KUKA KRL program: MyProgram_266().src

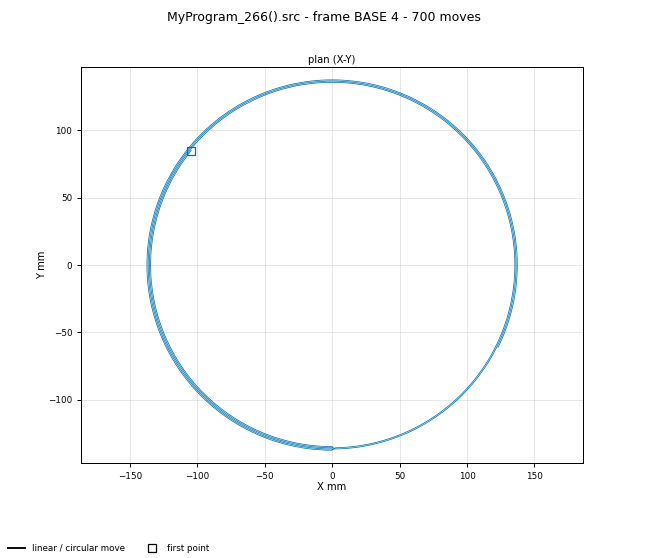
[picture p0: tool path of MyProgram_266().src in frame BASE 4, 700 of 700 moves have a stored position in this frame; points joined in program order, loops and branches not executed]
&ACCESS RVP
&REL 1
&PARAM TEMPLATE = C:\KRC\Roboter\Template\vorgabe
&PARAM EDITMASK = *
DEF MyProgram_266()
; ---- Setting reference (Base) ----
$BASE = BASE_DATA[4]

; --------------------------
; ---- Setting tool (TCP) ----
$TOOL = TOOL_DATA[3]
; --------------------------

$VEL.CP = VEL_APROX_PRINT
Startdeposition()
$VEL.CP = VEL_PRINT
LIN {X -104.4746,Y 84.848,Z 169,A 141.9621,B 9.8477,C 0.0918,E1 9.7233,E2 309.1377} C_DIS
LIN {X -107.2556,Y 81.3036,Z 169,A 143.6702,B 9.8476,C 0.1001,E1 9.7204,E2 307.4569} C_DIS
LIN {X -111.5663,Y 75.2791,Z 169,A 147.0659,B 9.8476,C 0.1033,E1 9.7149,E2 304.0355} C_DIS
LIN {X -114.0415,Y 71.475,Z 169,A 148.9826,B 9.8475,C 0.1084,E1 9.712,E2 302.1227} C_DIS
LIN {X -115.8284,Y 68.5413,Z 169,A 150.5259,B 9.8475,C 0.1107,E1 9.7098,E2 300.5712} C_DIS
LIN {X -118.6938,Y 63.4493,Z 169,A 153.1021,B 9.8474,C 0.1155,E1 9.7063,E2 297.9869} C_DIS
LIN {X -120.5086,Y 59.9271,Z 169,A 154.6631,B 9.8474,C 0.1222,E1 9.7043,E2 296.4429} C_DIS
LIN {X -122.0379,Y 56.7472,Z 169,A 156.1056,B 9.8473,C 0.1272,E1 9.7026,E2 295.0093} C_DIS
LIN {X -123.501,Y 53.4877,Z 169,A 157.6774,B 9.8473,C 0.1304,E1 9.7009,E2 293.4329} C_DIS
LIN {X -124.8461,Y 50.2682,Z 169,A 159.1832,B 9.8472,C 0.1341,E1 9.6993,E2 291.9263} C_DIS
LIN {X -126.2668,Y 46.5893,Z 169,A 161.0061,B 9.8472,C 0.1361,E1 9.6974,E2 290.0877} C_DIS
LIN {X -127.5662,Y 42.9007,Z 169,A 162.6082,B 9.8471,C 0.1419,E1 9.696,E2 288.495} C_DIS
LIN {X -128.6173,Y 39.6372,Z 169,A 164.0174,B 9.847,C 0.1468,E1 9.6948,E2 287.0935} C_DIS
LIN {X -129.8851,Y 35.2642,Z 169,A 166.1874,B 9.847,C 0.1482,E1 9.6932,E2 284.8975} C_DIS
LIN {X -130.8817,Y 31.3605,Z 169,A 168.0934,B 9.847,C 0.1497,E1 9.6919,E2 282.97} C_DIS
LIN {X -131.6037,Y 28.1781,Z 169,A 169.2729,B 9.8468,C 0.1574,E1 9.6912,E2 281.8174} C_DIS
LIN {X -132.3186,Y 24.6117,Z 169,A 171.627,B 9.847,C 0.1475,E1 9.69,E2 279.3666} C_DIS
LIN {X -133.2931,Y 18.6182,Z 169,A 173.4883,B 9.8466,C 0.1679,E1 9.6893,E2 277.5966} C_DIS
LIN {X -133.7452,Y 15.0386,Z 169,A 175.0197,B 9.8466,C 0.1725,E1 9.6887,E2 276.0674} C_DIS
LIN {X -134.1082,Y 11.3371,Z 169,A 176.5691,B 9.8465,C 0.1777,E1 9.6884,E2 274.5236} C_DIS
LIN {X -134.3787,Y 7.5153,Z 169,A 178.3708,B 9.8465,C 0.1794,E1 9.688,E2 272.7028} C_DIS
LIN {X -134.5281,Y 3.9764,Z 169,A 179.8134,B 9.8463,C 0.1849,E1 9.688,E2 271.2696} C_DIS
LIN {X -134.589,Y -0.2836,Z 169,A -178.249,B 9.8463,C 0.188,E1 9.6879,E2 269.3188} C_DIS
LIN {X -134.5104,Y -4.577,Z 169,A -176.4181,B 9.8462,C 0.1933,E1 9.688,E2 267.4893} C_DIS
LIN {X -134.2976,Y -8.8324,Z 169,A -174.5756,B 9.8461,C 0.1981,E1 9.6883,E2 265.6449} C_DIS
LIN {X -133.9649,Y -12.9206,Z 169,A -172.93,B 9.846,C 0.2049,E1 9.6887,E2 264.0132} C_DIS
LIN {X -133.5317,Y -16.8296,Z 169,A -171.2069,B 9.8459,C 0.2089,E1 9.6893,E2 262.2858} C_DIS
LIN {X -133.1154,Y -19.8582,Z 169,A -169.0696,B 9.8461,C 0.1976,E1 9.6903,E2 260.0468} C_DIS
LIN {X -132.0948,Y -25.7822,Z 169,A -167.1873,B 9.8457,C 0.2171,E1 9.6912,E2 258.2501} C_DIS
LIN {X -131.1442,Y -30.2452,Z 169,A -165.035,B 9.8457,C 0.2188,E1 9.6925,E2 256.0738} C_DIS
LIN {X -130.3652,Y -33.4442,Z 169,A -163.6911,B 9.8455,C 0.2238,E1 9.6934,E2 254.7381} C_DIS
LIN {X -129.1038,Y -38.0226,Z 169,A -161.8309,B 9.8454,C 0.2323,E1 9.6948,E2 252.8994} C_DIS
LIN {X -127.7896,Y -42.2298,Z 169,A -159.9505,B 9.8452,C 0.2374,E1 9.6964,E2 251.02} C_DIS
LIN {X -126.6409,Y -45.5579,Z 169,A -158.4535,B 9.8452,C 0.2415,E1 9.6978,E2 249.5244} C_DIS
LIN {X -125.6224,Y -48.298,Z 169,A -157.1558,B 9.8451,C 0.2439,E1 9.6991,E2 248.2211} C_DIS
LIN {X -124.3665,Y -51.4452,Z 169,A -155.6269,B 9.8451,C 0.2462,E1 9.7007,E2 246.6826} C_DIS
LIN {X -123.0232,Y -54.5791,Z 169,A -153.402,B 9.8453,C 0.2358,E1 9.7034,E2 244.363} C_DIS
LIN {X -120.4151,Y -60.1168,Z 169,A -151.6536,B 9.8447,C 0.2583,E1 9.7054,E2 242.7227} C_DIS
LIN {X -117.7451,Y -65.1924,Z 169,A -149.0637,B 9.8447,C 0.2617,E1 9.7088,E2 240.1161} C_DIS
LIN {X -115.6191,Y -68.8925,Z 169,A -147.1761,B 9.8445,C 0.2649,E1 9.7115,E2 238.2208} C_DIS
LIN {X -113.6955,Y -72.0231,Z 169,A -145.4698,B 9.8445,C 0.2661,E1 9.7141,E2 236.498} C_DIS
LIN {X -110.2679,Y -77.1691,Z 169,A -142.9073,B 9.8443,C 0.2735,E1 9.7181,E2 233.9455} C_DIS
LIN {X -108.3076,Y -79.8967,Z 169,A -141.4872,B 9.8443,C 0.277,E1 9.7204,E2 232.5274} C_DIS
LIN {X -105.6392,Y -83.3931,Z 169,A -139.5784,B 9.8441,C 0.2805,E1 9.7237,E2 230.615} C_DIS
LIN {X -102.9213,Y -86.7251,Z 169,A -137.755,B 9.844,C 0.2846,E1 9.7269,E2 228.7932} C_DIS
LIN {X -100.0131,Y -90.0636,Z 169,A -135.8758,B 9.8439,C 0.2887,E1 9.7304,E2 226.9156} C_DIS
LIN {X -97.1849,Y -93.1078,Z 169,A -134.0881,B 9.8438,C 0.292,E1 9.7338,E2 225.1263} C_DIS
LIN {X -94.1505,Y -96.1751,Z 169,A -132.2221,B 9.8437,C 0.295,E1 9.7375,E2 223.2573} C_DIS
LIN {X -90.8936,Y -99.2591,Z 169,A -130.2911,B 9.8436,C 0.2983,E1 9.7415,E2 221.3242} C_DIS
LIN {X -87.2585,Y -102.4691,Z 169,A -127.3053,B 9.844,C 0.2841,E1 9.7481,E2 218.2237} C_DIS
LIN {X -81.9586,Y -106.7557,Z 169,A -124.5269,B 9.8438,C 0.2915,E1 9.7542,E2 215.4616} C_DIS
LIN {X -77.0946,Y -110.3197,Z 169,A -122.6505,B 9.8433,C 0.3091,E1 9.7583,E2 213.6722} C_DIS
LIN {X -73.3974,Y -112.813,Z 169,A -120.7481,B 9.8432,C 0.3119,E1 9.7627,E2 211.7696} C_DIS
LIN {X -69.5467,Y -115.2268,Z 169,A -118.9875,B 9.843,C 0.3181,E1 9.7668,E2 210.0308} C_DIS
LIN {X -66.5586,Y -116.9783,Z 169,A -117.3469,B 9.843,C 0.3168,E1 9.7708,E2 208.3697} C_DIS
LIN {X -62.9884,Y -118.9373,Z 169,A -115.8149,B 9.8428,C 0.323,E1 9.7745,E2 206.8628} C_DIS
LIN {X -57.8669,Y -121.5107,Z 169,A -113.1985,B 9.8428,C 0.3224,E1 9.7812,E2 204.2246} C_DIS
LIN {X -54.566,Y -123.029,Z 169,A -111.6015,B 9.8428,C 0.3231,E1 9.7852,E2 202.6214} C_DIS
LIN {X -51.0188,Y -124.5433,Z 169,A -109.667,B 9.843,C 0.3189,E1 9.7903,E2 200.6502} C_DIS
LIN {X -47.8413,Y -125.797,Z 169,A -108.374,B 9.8428,C 0.3235,E1 9.7936,E2 199.3772} C_DIS
LIN {X -44.7366,Y -126.9352,Z 169,A -106.7852,B 9.8428,C 0.321,E1 9.7979,E2 197.7656} C_DIS
LIN {X -41.4449,Y -128.047,Z 169,A -105.5584,B 9.8427,C 0.3273,E1 9.8011,E2 196.5703} C_DIS
LIN {X -36.6892,Y -129.4897,Z 169,A -103.585,B 9.8425,C 0.3317,E1 9.8063,E2 194.6143} C_DIS
LIN {X -33.2756,Y -130.408,Z 169,A -101.9665,B 9.8425,C 0.3303,E1 9.8107,E2 192.9812} C_DIS
LIN {X -29.4826,Y -131.3183,Z 169,A -100.2296,B 9.8425,C 0.3296,E1 9.8155,E2 191.2344} C_DIS
LIN {X -25.4985,Y -132.149,Z 169,A -98.6989,B 9.8425,C 0.3346,E1 9.8196,E2 189.7285} C_DIS
LIN {X -22.0927,Y -132.7608,Z 169,A -97.1167,B 9.8425,C 0.3329,E1 9.824,E2 188.1322} C_DIS
LIN {X -17.9158,Y -133.3894,Z 169,A -95.3049,B 9.8425,C 0.3331,E1 9.829,E2 186.3181} C_DIS
LIN {X -14.222,Y -133.8331,Z 169,A -93.7187,B 9.8425,C 0.3334,E1 9.8334,E2 184.7311} C_DIS
LIN {X -9.9772,Y -134.2163,Z 169,A -91.8812,B 9.8425,C 0.3331,E1 9.8385,E2 182.8899} C_DIS
LIN {X -6.3934,Y -134.4352,Z 169,A -90.4095,B 9.8425,C 0.3344,E1 9.8426,E2 181.4247} C_DIS
LIN {X 0.0501,Y -134.5885,Z 169,A -87.5776,B 9.8425,C 0.3323,E1 9.8506,E2 178.5806} C_DIS
LIN {X 0.0501,Y -134.5885,Z 169,A -87.5776,B 9.8425,C 0.3323,E1 9.8506,E2 178.5806} C_DIS
Enddeposition()
LIN {X 0.9846,Y -135.4934,Z 169,A -87.3396,B 9.8083,C 0.3426,E1 9.8172,E2 178.4063} C_DIS
Startdeposition()
$VEL.CP = VEL_PRINT
LIN {X -1.7041,Y -135.4894,Z 169,A -89.4595,B 9.8075,C 0.3636,E1 9.8109,E2 180.6497} C_DIS
LIN {X -5.8269,Y -135.3747,Z 169,A -91.2545,B 9.8075,C 0.3647,E1 9.8059,E2 182.4517} C_DIS
LIN {X -10.1659,Y -135.1174,Z 169,A -92.6919,B 9.8078,C 0.3562,E1 9.802,E2 183.8402} C_DIS
LIN {X -14.3572,Y -134.7362,Z 169,A -94.441,B 9.8078,C 0.3552,E1 9.7972,E2 185.5862} C_DIS
LIN {X -18.8026,Y -134.1884,Z 169,A -96.1751,B 9.808,C 0.3514,E1 9.7924,E2 187.301} C_DIS
LIN {X -22.1311,Y -133.6793,Z 169,A -97.7451,B 9.8079,C 0.354,E1 9.788,E2 188.8897} C_DIS
LIN {X -26.262,Y -132.9316,Z 169,A -99.5573,B 9.8079,C 0.354,E1 9.783,E2 190.707} C_DIS
LIN {X -30.094,Y -132.1145,Z 169,A -101.001,B 9.8081,C 0.3488,E1 9.7792,E2 192.1245} C_DIS
LIN {X -32.876,Y -131.4507,Z 169,A -102.333,B 9.8081,C 0.3506,E1 9.7755,E2 193.4722} C_DIS
LIN {X -36.2856,Y -130.5499,Z 169,A -103.8661,B 9.8081,C 0.3506,E1 9.7714,E2 195.0107} C_DIS
LIN {X -39.7461,Y -129.5381,Z 169,A -105.3796,B 9.8081,C 0.3492,E1 9.7673,E2 196.5231} C_DIS
LIN {X -42.9923,Y -128.4973,Z 169,A -107.0189,B 9.808,C 0.3521,E1 9.7629,E2 198.1872} C_DIS
LIN {X -47.0136,Y -127.0821,Z 169,A -108.6772,B 9.8081,C 0.3476,E1 9.7586,E2 199.8278} C_DIS
LIN {X -52.4076,Y -124.9533,Z 169,A -111.1063,B 9.8082,C 0.3447,E1 9.7523,E2 202.2542} C_DIS
LIN {X -55.9076,Y -123.4284,Z 169,A -112.7383,B 9.8082,C 0.3434,E1 9.7481,E2 203.8885} C_DIS
LIN {X -59.6258,Y -121.6746,Z 169,A -114.6061,B 9.8082,C 0.3439,E1 9.7434,E2 205.7723} C_DIS
LIN {X -63.9943,Y -119.4367,Z 169,A -116.6408,B 9.8084,C 0.3405,E1 9.7384,E2 207.8019} C_DIS
LIN {X -67.9227,Y -117.2471,Z 169,A -118.5074,B 9.8084,C 0.3373,E1 9.7339,E2 209.6641} C_DIS
LIN {X -71.4696,Y -115.1194,Z 169,A -120.3282,B 9.8085,C 0.3362,E1 9.7295,E2 211.4936} C_DIS
LIN {X -75.3032,Y -112.649,Z 169,A -122.2736,B 9.8085,C 0.3337,E1 9.7249,E2 213.4408} C_DIS
LIN {X -78.9155,Y -110.1486,Z 169,A -124.3329,B 9.8085,C 0.3346,E1 9.7202,E2 215.5246} C_DIS
LIN {X -81.4969,Y -108.2527,Z 169,A -125.5133,B 9.8087,C 0.329,E1 9.7176,E2 216.6833} C_DIS
LIN {X -85.0693,Y -105.4684,Z 169,A -127.7248,B 9.8087,C 0.3314,E1 9.7127,E2 218.9308} C_DIS
LIN {X -87.918,Y -103.1059,Z 169,A -129.0319,B 9.8089,C 0.3237,E1 9.71,E2 220.2058} C_DIS
LIN {X -91.3335,Y -100.0935,Z 169,A -130.9853,B 9.809,C 0.3206,E1 9.7059,E2 222.1621} C_DIS
LIN {X -94.519,Y -97.091,Z 169,A -132.8484,B 9.8091,C 0.3173,E1 9.7021,E2 224.0261} C_DIS
LIN {X -97.6402,Y -93.9517,Z 169,A -134.7461,B 9.8092,C 0.314,E1 9.6984,E2 225.9263} C_DIS
LIN {X -100.7027,Y -90.6612,Z 169,A -136.6867,B 9.8093,C 0.3108,E1 9.6948,E2 227.871} C_DIS
LIN {X -103.774,Y -87.1282,Z 169,A -138.6415,B 9.8095,C 0.3061,E1 9.6912,E2 229.8219} C_DIS
LIN {X -106.6225,Y -83.6182,Z 169,A -140.56,B 9.8096,C 0.302,E1 9.6879,E2 231.7404} C_DIS
LIN {X -108.5995,Y -81.0341,Z 169,A -142.1183,B 9.8096,C 0.3022,E1 9.6852,E2 233.3204} C_DIS
LIN {X -114.4696,Y -72.5061,Z 169,A -146.4334,B 9.8099,C 0.2908,E1 9.6785,E2 237.6255} C_DIS
LIN {X -116.9185,Y -68.487,Z 169,A -148.4029,B 9.8101,C 0.2855,E1 9.6757,E2 239.5912} C_DIS
LIN {X -118.9187,Y -64.9516,Z 169,A -150.3114,B 9.8101,C 0.2847,E1 9.6731,E2 241.522} C_DIS
LIN {X -121.339,Y -60.3062,Z 169,A -152.1729,B 9.8105,C 0.2726,E1 9.6708,E2 243.3388} C_DIS
LIN {X -122.6794,Y -57.5337,Z 169,A -153.9307,B 9.8103,C 0.2775,E1 9.6686,E2 245.1515} C_DIS
LIN {X -124.0401,Y -54.5398,Z 169,A -155.1704,B 9.8105,C 0.2712,E1 9.6672,E2 246.3718} C_DIS
LIN {X -125.5769,Y -50.8953,Z 169,A -156.597,B 9.8107,C 0.2623,E1 9.6657,E2 247.767} C_DIS
LIN {X -126.8021,Y -47.7612,Z 169,A -158.2342,B 9.8107,C 0.2623,E1 9.6641,E2 249.4295} C_DIS
LIN {X -127.9517,Y -44.5899,Z 169,A -159.6507,B 9.8108,C 0.2583,E1 9.6627,E2 250.8436} C_DIS
LIN {X -129.019,Y -41.4004,Z 169,A -161.047,B 9.811,C 0.2539,E1 9.6615,E2 252.2356} C_DIS
LIN {X -130.5089,Y -36.4323,Z 169,A -163.11,B 9.8112,C 0.2455,E1 9.6599,E2 254.281} C_DIS
LIN {X -131.8344,Y -31.3017,Z 169,A -165.6779,B 9.8112,C 0.2451,E1 9.6581,E2 256.8871} C_DIS
LIN {X -132.6884,Y -27.4572,Z 169,A -167.2993,B 9.8113,C 0.2396,E1 9.6572,E2 258.5018} C_DIS
LIN {X -133.2596,Y -24.5412,Z 169,A -168.4771,B 9.8114,C 0.2346,E1 9.6566,E2 259.6689} C_DIS
LIN {X -134.0173,Y -19.9962,Z 169,A -170.6665,B 9.8114,C 0.2333,E1 9.6556,E2 261.8859} C_DIS
LIN {X -134.5452,Y -16.0475,Z 169,A -172.265,B 9.8116,C 0.2269,E1 9.655,E2 263.4724} C_DIS
LIN {X -134.9764,Y -11.8982,Z 169,A -174.0668,B 9.8117,C 0.2225,E1 9.6545,E2 265.2772} C_DIS
LIN {X -135.249,Y -8.2276,Z 169,A -175.6609,B 9.8117,C 0.2186,E1 9.6542,E2 266.8744} C_DIS
LIN {X -135.4408,Y -3.9755,Z 169,A -177.3758,B 9.8119,C 0.2119,E1 9.6541,E2 268.5773} C_DIS
LIN {X -135.4946,Y -1.2451,Z 169,A -178.5875,B 9.8119,C 0.2095,E1 9.6541,E2 269.7948} C_DIS
LIN {X -135.4778,Y 2.4043,Z 169,A 179.802,B 9.8121,C 0.2062,E1 9.6541,E2 271.412} C_DIS
LIN {X -135.3439,Y 6.4888,Z 169,A 178.0277,B 9.8121,C 0.202,E1 9.6543,E2 273.1901} C_DIS
LIN {X -135.0971,Y 10.4433,Z 169,A 176.2627,B 9.8122,C 0.1987,E1 9.6546,E2 274.9644} C_DIS
LIN {X -134.7164,Y 14.541,Z 169,A 174.6123,B 9.8123,C 0.192,E1 9.6551,E2 276.6021} C_DIS
LIN {X -134.3046,Y 17.9539,Z 169,A 173.0148,B 9.8123,C 0.1904,E1 9.6556,E2 278.2155} C_DIS
LIN {X -133.5133,Y 23.1204,Z 169,A 170.7631,B 9.8125,C 0.1847,E1 9.6566,E2 280.47} C_DIS
LIN {X -132.7842,Y 26.9862,Z 169,A 169.1918,B 9.8126,C 0.1783,E1 9.6575,E2 282.0284} C_DIS
LIN {X -132.0036,Y 30.5797,Z 169,A 167.3619,B 9.8126,C 0.1787,E1 9.6586,E2 283.8898} C_DIS
LIN {X -130.7428,Y 35.5906,Z 169,A 165.5062,B 9.8128,C 0.1667,E1 9.6599,E2 285.7036} C_DIS
LIN {X -129.6128,Y 39.5021,Z 169,A 163.6634,B 9.8128,C 0.164,E1 9.6614,E2 287.5591} C_DIS
LIN {X -128.6362,Y 42.5751,Z 169,A 162.3969,B 9.8129,C 0.1585,E1 9.6624,E2 288.8125} C_DIS
LIN {X -127.6556,Y 45.4337,Z 169,A 160.8869,B 9.8129,C 0.159,E1 9.6638,E2 290.3491} C_DIS
LIN {X -126.4641,Y 48.6508,Z 169,A 159.4229,B 9.8129,C 0.1553,E1 9.6653,E2 291.8133} C_DIS
LIN {X -125.1301,Y 51.9841,Z 169,A 158.0209,B 9.8131,C 0.1491,E1 9.6667,E2 293.1996} C_DIS
LIN {X -123.8888,Y 54.8783,Z 169,A 156.7323,B 9.8131,C 0.1448,E1 9.6682,E2 294.4816} C_DIS
LIN {X -122.3782,Y 58.1677,Z 169,A 154.9956,B 9.8131,C 0.1443,E1 9.6702,E2 296.2415} C_DIS
LIN {X -120.8397,Y 61.2994,Z 169,A 153.5628,B 9.8132,C 0.1397,E1 9.672,E2 297.6676} C_DIS
LIN {X -119.2264,Y 64.3856,Z 169,A 151.7311,B 9.8132,C 0.1422,E1 9.6745,E2 299.5409} C_DIS
LIN {X -117.537,Y 67.4206,Z 169,A 150.5451,B 9.8133,C 0.1335,E1 9.6761,E2 300.6914} C_DIS
LIN {X -115.4093,Y 71.0006,Z 169,A 148.7054,B 9.8133,C 0.1304,E1 9.6788,E2 302.5387} C_DIS
LIN {X -113.1396,Y 74.5641,Z 169,A 146.8982,B 9.8134,C 0.1264,E1 9.6815,E2 304.3465} C_DIS
LIN {X -110.8638,Y 77.9079,Z 169,A 144.9205,B 9.8134,C 0.127,E1 9.6847,E2 306.3544} C_DIS
LIN {X -108.8461,Y 80.703,Z 169,A 143.6604,B 9.8134,C 0.12,E1 9.6867,E2 307.5893} C_DIS
LIN {X -106.124,Y 84.2501,Z 169,A 141.7568,B 9.8135,C 0.1158,E1 9.69,E2 309.4925} C_DIS
LIN {X -103.3075,Y 87.6809,Z 169,A 139.7708,B 9.8135,C 0.1136,E1 9.6936,E2 311.4895} C_DIS
LIN {X -100.8359,Y 90.5125,Z 169,A 137.7323,B 9.8135,C 0.1182,E1 9.6975,E2 313.5799} C_DIS
LIN {X -97.4544,Y 94.1436,Z 169,A 136.1412,B 9.8137,C 0.1045,E1 9.7004,E2 315.1086} C_DIS
LIN {X -94.3245,Y 97.2792,Z 169,A 134.5267,B 9.8137,C 0.0959,E1 9.7036,E2 316.6901} C_DIS
LIN {X -92.0472,Y 99.4376,Z 169,A 132.1572,B 9.8136,C 0.1122,E1 9.7087,E2 319.1826} C_DIS
LIN {X -87.4769,Y 103.4809,Z 169,A 130.2745,B 9.8138,C 0.0945,E1 9.7125,E2 320.98} C_DIS
LIN {X -83.9845,Y 106.3349,Z 169,A 128.4876,B 9.8138,C 0.0887,E1 9.7163,E2 322.7507} C_DIS
LIN {X -80.3236,Y 109.126,Z 169,A 126.3949,B 9.8138,C 0.088,E1 9.7211,E2 324.859} C_DIS
LIN {X -76.8138,Y 111.6245,Z 169,A 124.5797,B 9.8138,C 0.0848,E1 9.7252,E2 326.6717} C_DIS
LIN {X -73.3748,Y 113.9151,Z 169,A 122.8281,B 9.8138,C 0.082,E1 9.7293,E2 328.4223} C_DIS
LIN {X -69.9245,Y 116.0645,Z 169,A 121.1217,B 9.8138,C 0.0791,E1 9.7333,E2 330.1257} C_DIS
LIN {X -65.3863,Y 118.6806,Z 169,A 118.9507,B 9.8139,C 0.075,E1 9.7386,E2 332.2895} C_DIS
LIN {X -56.3707,Y 123.2172,Z 169,A 114.5055,B 9.8139,C 0.0728,E1 9.7498,E2 336.7524} C_DIS
LIN {X -52.5239,Y 124.9047,Z 169,A 112.9588,B 9.8139,C 0.0662,E1 9.7537,E2 338.2702} C_DIS
LIN {X -48.3408,Y 126.5842,Z 169,A 110.5266,B 9.8139,C 0.0743,E1 9.7601,E2 340.7639} C_DIS
LIN {X -44.8214,Y 127.8715,Z 169,A 109.2132,B 9.8139,C 0.0674,E1 9.7635,E2 342.0437} C_DIS
LIN {X -40.9973,Y 129.1478,Z 169,A 107.5943,B 9.814,C 0.0642,E1 9.7678,E2 343.651} C_DIS
LIN {X -37.8633,Y 130.1011,Z 169,A 105.8355,B 9.814,C 0.0703,E1 9.7726,E2 345.4535} C_DIS
LIN {X -34.0681,Y 131.1481,Z 169,A 104.397,B 9.814,C 0.0646,E1 9.7764,E2 346.864} C_DIS
LIN {X -30.3036,Y 132.0667,Z 169,A 102.9781,B 9.814,C 0.0591,E1 9.7802,E2 348.2555} C_DIS
LIN {X -27.3014,Y 132.7201,Z 169,A 101.5914,B 9.814,C 0.06,E1 9.784,E2 349.6517} C_DIS
LIN {X -23.9521,Y 133.365,Z 169,A 100.0983,B 9.814,C 0.0602,E1 9.7881,E2 351.15} C_DIS
LIN {X -19.7291,Y 134.056,Z 169,A 98.2965,B 9.814,C 0.0592,E1 9.7931,E2 352.9499} C_DIS
LIN {X -16.1448,Y 134.5336,Z 169,A 96.9592,B 9.814,C 0.0547,E1 9.7967,E2 354.2633} C_DIS
LIN {X -13.4132,Y 134.8342,Z 169,A 95.7974,B 9.814,C 0.0543,E1 9.8,E2 355.4244} C_DIS
LIN {X -9.9919,Y 135.1301,Z 169,A 94.1589,B 9.814,C 0.0577,E1 9.8046,E2 357.0844} C_DIS
LIN {X -5.836,Y 135.3744,Z 169,A 92.3544,B 9.814,C 0.0583,E1 9.8096,E2 358.8934} C_DIS
LIN {X -2.5296,Y 135.4757,Z 169,A 91.0733,B 9.814,C 0.0557,E1 9.8132,E2 360.1598} C_DIS
LIN {X 0.959,Y 135.4958,Z 169,A 89.4469,B 9.814,C 0.0588,E1 9.8178,E2 361.8035} C_DIS
LIN {X 5.1409,Y 135.4015,Z 169,A 87.7755,B 9.814,C 0.0568,E1 9.8224,E2 363.4625} C_DIS
LIN {X 8.9955,Y 135.2016,Z 169,A 86.048,B 9.814,C 0.0591,E1 9.8272,E2 365.2009} C_DIS
LIN {X 12.6129,Y 134.911,Z 169,A 84.6543,B 9.814,C 0.0565,E1 9.8311,E2 366.5771} C_DIS
LIN {X 16.0427,Y 134.5458,Z 169,A 83.168,B 9.814,C 0.0575,E1 9.8352,E2 368.0661} C_DIS
LIN {X 20.1948,Y 133.9865,Z 169,A 81.3304,B 9.814,C 0.0595,E1 9.8403,E2 369.9112} C_DIS
LIN {X 23.8243,Y 133.3878,Z 169,A 79.8898,B 9.814,C 0.0578,E1 9.8442,E2 371.3375} C_DIS
LIN {X 27.1331,Y 132.7543,Z 169,A 78.4485,B 9.814,C 0.0589,E1 9.8482,E2 372.7805} C_DIS
LIN {X 30.0069,Y 132.1344,Z 169,A 77.1946,B 9.814,C 0.0599,E1 9.8516,E2 374.0353} C_DIS
LIN {X 33.3964,Y 131.3186,Z 169,A 75.746,B 9.814,C 0.0603,E1 9.8555,E2 375.4805} C_DIS
LIN {X 37.0587,Y 130.3337,Z 169,A 74.0247,B 9.814,C 0.064,E1 9.8602,E2 377.2157} C_DIS
LIN {X 42.0503,Y 128.811,Z 169,A 71.8034,B 9.814,C 0.0662,E1 9.8661,E2 379.4386} C_DIS
LIN {X 45.2991,Y 127.7041,Z 169,A 70.5454,B 9.814,C 0.0634,E1 9.8694,E2 380.6731} C_DIS
LIN {X 50.0829,Y 125.9044,Z 169,A 68.2517,B 9.814,C 0.0684,E1 9.8754,E2 382.9825} C_DIS
LIN {X 53.5446,Y 124.4704,Z 169,A 66.8073,B 9.814,C 0.0671,E1 9.8791,E2 384.41} C_DIS
LIN {X 56.4831,Y 123.1652,Z 169,A 65.571,B 9.814,C 0.066,E1 9.8822,E2 385.6313} C_DIS
LIN {X 58.8241,Y 122.0646,Z 169,A 64.2048,B 9.814,C 0.0733,E1 9.8857,E2 387.0305} C_DIS
LIN {X 62.1857,Y 120.3885,Z 169,A 62.6394,B 9.814,C 0.0749,E1 9.8896,E2 388.5932} C_DIS
LIN {X 65.9948,Y 118.3437,Z 169,A 60.8518,B 9.814,C 0.0765,E1 9.894,E2 390.376} C_DIS
LIN {X 71.1606,Y 115.3111,Z 169,A 58.3825,B 9.8139,C 0.0788,E1 9.8999,E2 392.8379} C_DIS
LIN {X 74.674,Y 113.0672,Z 169,A 56.7523,B 9.8139,C 0.0785,E1 9.9036,E2 394.4523} C_DIS
LIN {X 77.9743,Y 110.8169,Z 169,A 54.9437,B 9.8139,C 0.084,E1 9.9078,E2 396.2757} C_DIS
LIN {X 80.3443,Y 109.1109,Z 169,A 53.721,B 9.8139,C 0.0858,E1 9.9106,E2 397.4971} C_DIS
LIN {X 82.9656,Y 107.1311,Z 169,A 52.2684,B 9.8139,C 0.0896,E1 9.9138,E2 398.9577} C_DIS
LIN {X 86.5459,Y 104.2602,Z 169,A 50.3901,B 9.8138,C 0.0917,E1 9.9179,E2 400.829} C_DIS
LIN {X 90.0068,Y 101.288,Z 169,A 48.5146,B 9.8138,C 0.0941,E1 9.9218,E2 402.6985} C_DIS
LIN {X 93.1652,Y 98.3904,Z 169,A 46.6712,B 9.8138,C 0.0984,E1 9.9256,E2 404.5463} C_DIS
LIN {X 96.3812,Y 95.2427,Z 169,A 44.8099,B 9.8137,C 0.1013,E1 9.9293,E2 406.4033} C_DIS
LIN {X 99.3958,Y 92.0921,Z 169,A 42.985,B 9.8137,C 0.1047,E1 9.9328,E2 408.2266} C_DIS
LIN {X 102.3394,Y 88.8096,Z 169,A 41.103,B 9.8137,C 0.1091,E1 9.9362,E2 410.1116} C_DIS
LIN {X 105.1031,Y 85.5207,Z 169,A 39.4275,B 9.8136,C 0.1099,E1 9.9392,E2 411.7706} C_DIS
LIN {X 107.5253,Y 82.4543,Z 169,A 37.6875,B 9.8136,C 0.1157,E1 9.9422,E2 413.5221} C_DIS
LIN {X 110.1599,Y 78.8997,Z 169,A 35.8884,B 9.8136,C 0.1183,E1 9.9452,E2 415.3134} C_DIS
LIN {X 112.612,Y 75.3587,Z 169,A 34.0464,B 9.8134,C 0.1232,E1 9.9481,E2 417.159} C_DIS
LIN {X 115.0806,Y 71.532,Z 169,A 32.1983,B 9.8134,C 0.126,E1 9.9508,E2 418.9987} C_DIS
LIN {X 117.2434,Y 67.929,Z 169,A 29.9628,B 9.8132,C 0.1412,E1 9.954,E2 421.2909} C_DIS
LIN {X 119.4402,Y 63.9877,Z 169,A 28.466,B 9.8132,C 0.1364,E1 9.956,E2 422.7391} C_DIS
LIN {X 121.5411,Y 59.8964,Z 169,A 26.6662,B 9.8132,C 0.138,E1 9.9582,E2 424.5223} C_DIS
LIN {X 123.1884,Y 56.433,Z 169,A 24.9613,B 9.8132,C 0.1442,E1 9.9602,E2 426.2385} C_DIS
LIN {X 125.0293,Y 52.2256,Z 169,A 23.2463,B 9.8132,C 0.144,E1 9.9621,E2 427.9272} C_DIS
LIN {X 126.231,Y 49.2504,Z 169,A 21.3562,B 9.8129,C 0.1603,E1 9.9641,E2 429.8834} C_DIS
LIN {X 127.7616,Y 45.1382,Z 169,A 19.8812,B 9.8129,C 0.1563,E1 9.9654,E2 431.3134} C_DIS
LIN {X 129.9739,Y 38.2978,Z 169,A 16.97,B 9.8129,C 0.1617,E1 9.9679,E2 434.2113} C_DIS
LIN {X 130.9481,Y 34.8209,Z 169,A 15.4742,B 9.8129,C 0.1652,E1 9.969,E2 435.7045} C_DIS
LIN {X 131.9527,Y 30.8026,Z 169,A 13.6603,B 9.8127,C 0.1716,E1 9.9702,E2 437.5275} C_DIS
LIN {X 132.7658,Y 27.0768,Z 169,A 12.1863,B 9.8127,C 0.1729,E1 9.971,E2 438.9859} C_DIS
LIN {X 133.4044,Y 23.7316,Z 169,A 10.7148,B 9.8127,C 0.1777,E1 9.9718,E2 440.4625} C_DIS
LIN {X 134.1185,Y 19.2916,Z 169,A 8.8839,B 9.8125,C 0.1815,E1 9.9725,E2 442.2864} C_DIS
LIN {X 134.523,Y 16.2335,Z 169,A 7.5986,B 9.8125,C 0.1848,E1 9.973,E2 443.5705} C_DIS
LIN {X 134.9077,Y 12.6476,Z 169,A 6.0017,B 9.8124,C 0.191,E1 9.9734,E2 445.1777} C_DIS
LIN {X 135.2436,Y 8.3139,Z 169,A 4.2367,B 9.8123,C 0.1945,E1 9.9738,E2 446.9354} C_DIS
LIN {X 135.4292,Y 4.3942,Z 169,A 2.5722,B 9.8123,C 0.1995,E1 9.974,E2 448.6022} C_DIS
LIN {X 135.5028,Y -0.084,Z 169,A 0.6302,B 9.8121,C 0.2062,E1 9.974,E2 450.5521} C_DIS
LIN {X 135.4415,Y -3.9507,Z 169,A -0.8831,B 9.8121,C 0.208,E1 9.974,E2 452.0518} C_DIS
LIN {X 135.2471,Y -8.2574,Z 169,A -2.6483,B 9.8119,C 0.212,E1 9.9737,E2 453.8117} C_DIS
LIN {X 134.9316,Y -12.3986,Z 169,A -4.3806,B 9.8119,C 0.2165,E1 9.9733,E2 455.5428} C_DIS
LIN {X 134.5559,Y -15.9578,Z 169,A -5.851,B 9.8118,C 0.2199,E1 9.9728,E2 457.0094} C_DIS
LIN {X 134.0747,Y -19.5982,Z 169,A -7.4832,B 9.8116,C 0.2263,E1 9.9722,E2 458.653} C_DIS
LIN {X 133.4121,Y -23.689,Z 169,A -9.0862,B 9.8116,C 0.2278,E1 9.9714,E2 460.2393} C_DIS
LIN {X 132.8838,Y -26.497,Z 169,A -10.3699,B 9.8115,C 0.2331,E1 9.9707,E2 461.5337} C_DIS
LIN {X 132.1039,Y -30.1405,Z 169,A -11.8064,B 9.8115,C 0.2342,E1 9.9699,E2 462.9546} C_DIS
LIN {X 131.4138,Y -33.0214,Z 169,A -12.955,B 9.8115,C 0.2353,E1 9.9691,E2 464.0917} C_DIS
LIN {X 130.4064,Y -36.7987,Z 169,A -14.6657,B 9.8113,C 0.2414,E1 9.9679,E2 465.8113} C_DIS
LIN {X 129.42,Y -40.132,Z 169,A -16.2587,B 9.8111,C 0.2485,E1 9.9666,E2 467.4211} C_DIS
LIN {X 128.1467,Y -44.0274,Z 169,A -17.7218,B 9.8111,C 0.2468,E1 9.9653,E2 468.8525} C_DIS
LIN {X 127.3271,Y -46.3446,Z 169,A -19.0215,B 9.8109,C 0.256,E1 9.964,E2 470.1857} C_DIS
LIN {X 125.7603,Y -50.4404,Z 169,A -20.7135,B 9.8109,C 0.2572,E1 9.9623,E2 471.8596} C_DIS
LIN {X 124.5744,Y -53.3041,Z 169,A -22.0045,B 9.8108,C 0.2603,E1 9.9609,E2 473.1495} C_DIS
LIN {X 123.4317,Y -55.9003,Z 169,A -23.514,B 9.8105,C 0.271,E1 9.9592,E2 474.6988} C_DIS
LIN {X 121.9232,Y -59.12,Z 169,A -24.723,B 9.8105,C 0.268,E1 9.9577,E2 475.873} C_DIS
LIN {X 120.1324,Y -62.6749,Z 169,A -26.3419,B 9.8105,C 0.2709,E1 9.9557,E2 477.4857} C_DIS
LIN {X 117.8869,Y -66.8071,Z 169,A -28.6207,B 9.8102,C 0.283,E1 9.9525,E2 479.8027} C_DIS
LIN {X 116.1253,Y -69.824,Z 169,A -29.8713,B 9.8102,C 0.2814,E1 9.9508,E2 481.0268} C_DIS
LIN {X 113.7284,Y -73.663,Z 169,A -31.7289,B 9.8102,C 0.2848,E1 9.948,E2 482.8795} C_DIS
LIN {X 111.2085,Y -77.4147,Z 169,A -33.6802,B 9.8099,C 0.2905,E1 9.9449,E2 484.8379} C_DIS
LIN {X 108.4212,Y -81.2735,Z 169,A -35.4884,B 9.8099,C 0.2905,E1 9.942,E2 486.6227} C_DIS
LIN {X 105.9554,Y -84.462,Z 169,A -37.2508,B 9.8098,C 0.2959,E1 9.9389,E2 488.3941} C_DIS
LIN {X 103.8775,Y -87.0048,Z 169,A -38.6671,B 9.8097,C 0.2998,E1 9.9364,E2 489.8153} C_DIS
LIN {X 100.957,Y -90.3772,Z 169,A -40.523,B 9.8096,C 0.3034,E1 9.933,E2 491.6694} C_DIS
LIN {X 97.8292,Y -93.7541,Z 169,A -42.4274,B 9.8095,C 0.3067,E1 9.9293,E2 493.5706} C_DIS
LIN {X 95.3154,Y -96.3089,Z 169,A -43.9509,B 9.8094,C 0.3101,E1 9.9263,E2 495.0967} C_DIS
LIN {X 92.148,Y -99.3438,Z 169,A -45.7028,B 9.8094,C 0.3116,E1 9.9228,E2 496.8376} C_DIS
LIN {X 89.3297,Y -101.8856,Z 169,A -47.3697,B 9.8092,C 0.3163,E1 9.9193,E2 498.5139} C_DIS
LIN {X 86.0352,Y -104.6826,Z 169,A -49.1937,B 9.809,C 0.3198,E1 9.9154,E2 500.3392} C_DIS
LIN {X 82.2665,Y -107.6689,Z 169,A -51.1731,B 9.809,C 0.3223,E1 9.911,E2 502.3138} C_DIS
LIN {X 78.7716,Y -110.2515,Z 169,A -52.7931,B 9.809,C 0.3206,E1 9.9074,E2 503.9085} C_DIS
LIN {X 75.829,Y -112.2958,Z 169,A -54.5091,B 9.8088,C 0.3279,E1 9.9034,E2 505.6511} C_DIS
LIN {X 72.0718,Y -114.7437,Z 169,A -56.4,B 9.8087,C 0.331,E1 9.899,E2 507.543} C_DIS
LIN {X 67.1591,Y -117.6861,Z 169,A -58.806,B 9.8086,C 0.3345,E1 9.8932,E2 509.9493} C_DIS
LIN {X 63.2811,Y -119.8141,Z 169,A -60.4858,B 9.8086,C 0.3329,E1 9.8891,E2 511.6068} C_DIS
LIN {X 60.3553,Y -121.3147,Z 169,A -61.7893,B 9.8086,C 0.3329,E1 9.8859,E2 512.9007} C_DIS
LIN {X 57.2786,Y -122.7974,Z 169,A -63.566,B 9.8083,C 0.3424,E1 9.8813,E2 514.7202} C_DIS
LIN {X 52.714,Y -124.8253,Z 169,A -65.5199,B 9.8083,C 0.3415,E1 9.8763,E2 516.656} C_DIS
LIN {X 48.6765,Y -126.4541,Z 169,A -67.4042,B 9.8083,C 0.3447,E1 9.8714,E2 518.5473} C_DIS
LIN {X 45.2469,Y -127.7229,Z 169,A -68.9787,B 9.8081,C 0.347,E1 9.8673,E2 520.1266} C_DIS
LIN {X 41.267,Y -129.0616,Z 169,A -70.5536,B 9.8082,C 0.3444,E1 9.8631,E2 521.6777} C_DIS
LIN {X 38.4857,Y -129.9189,Z 169,A -71.8584,B 9.8082,C 0.3472,E1 9.8596,E2 522.9927} C_DIS
LIN {X 35.0276,Y -130.8929,Z 169,A -73.1634,B 9.8082,C 0.3438,E1 9.8562,E2 524.2719} C_DIS
LIN {X 31.9487,Y -131.6784,Z 169,A -74.7198,B 9.808,C 0.3497,E1 9.8519,E2 525.8559} C_DIS
LIN {X 28.3679,Y -132.4961,Z 169,A -76.292,B 9.808,C 0.3512,E1 9.8476,E2 527.4315} C_DIS
LIN {X 24.1233,Y -133.3343,Z 169,A -78.0006,B 9.808,C 0.3498,E1 9.843,E2 529.1262} C_DIS
LIN {X 21.2767,Y -133.819,Z 169,A -79.3442,B 9.808,C 0.3532,E1 9.8392,E2 530.486} C_DIS
LIN {X 17.0747,Y -134.4198,Z 169,A -81.1712,B 9.8079,C 0.3548,E1 9.8341,E2 532.318} C_DIS
LIN {X 12.9932,Y -134.8745,Z 169,A -82.7426,B 9.8079,C 0.352,E1 9.8298,E2 533.8698} C_DIS
LIN {X 9.8279,Y -135.142,Z 169,A -84.1232,B 9.8079,C 0.3533,E1 9.826,E2 535.2558} C_DIS
LIN {X 5.8603,Y -135.3734,Z 169,A -85.7549,B 9.8079,C 0.3527,E1 9.8214,E2 536.8823} C_DIS
LIN {X 2.4938,Y -135.4763,Z 169,A -87.2672,B 9.8079,C 0.3549,E1 9.8172,E2 538.4063} C_DIS
LIN {X 2.4938,Y -135.4763,Z 169,A -87.2672,B 9.8079,C 0.3549,E1 9.8172,E2 538.4063} C_DIS
Enddeposition()
LIN {X 0.9918,Y -136.4057,Z 169,A -87.4762,B 9.7767,C 0.3526,E1 9.7854,E2 538.6056} C_DIS
Startdeposition()
$VEL.CP = VEL_PRINT
LIN {X 3.4212,Y -136.3689,Z 169,A -86.3469,B 9.7768,C 0.3501,E1 9.7886,E2 537.4621} C_DIS
LIN {X 6.4779,Y -136.2579,Z 169,A -84.9138,B 9.7769,C 0.3466,E1 9.7927,E2 536.0095} C_DIS
LIN {X 9.5579,Y -136.0765,Z 169,A -83.7675,B 9.7769,C 0.3494,E1 9.7958,E2 534.8815} C_DIS
LIN {X 12.2574,Y -135.8617,Z 169,A -82.3457,B 9.7771,C 0.3428,E1 9.7999,E2 533.4229} C_DIS
LIN {X 15.844,Y -135.4883,Z 169,A -81.1431,B 9.7768,C 0.349,E1 9.8031,E2 532.2591} C_DIS
LIN {X 18.5107,Y -135.1517,Z 169,A -79.8391,B 9.777,C 0.3446,E1 9.8068,E2 530.9323} C_DIS
LIN {X 21.6604,Y -134.6828,Z 169,A -78.5032,B 9.777,C 0.3438,E1 9.8105,E2 529.5957} C_DIS
LIN {X 25.2313,Y -134.0579,Z 169,A -77.1382,B 9.777,C 0.3464,E1 9.8142,E2 528.2498} C_DIS
LIN {X 28.4035,Y -133.4218,Z 169,A -75.6268,B 9.777,C 0.342,E1 9.8184,E2 526.7181} C_DIS
LIN {X 31.7635,Y -132.6616,Z 169,A -74.2329,B 9.777,C 0.342,E1 9.8221,E2 525.3299} C_DIS
LIN {X 34.7637,Y -131.9076,Z 169,A -72.888,B 9.7772,C 0.3399,E1 9.8258,E2 523.9783} C_DIS
LIN {X 37.7611,Y -131.0817,Z 169,A -71.6108,B 9.7772,C 0.3394,E1 9.8292,E2 522.7038} C_DIS
LIN {X 40.7816,Y -130.1744,Z 169,A -70.2929,B 9.7772,C 0.3382,E1 9.8327,E2 521.3858} C_DIS
LIN {X 44.3,Y -129.0179,Z 169,A -68.7175,B 9.7772,C 0.3362,E1 9.8369,E2 519.8067} C_DIS
LIN {X 47.4655,Y -127.8871,Z 169,A -67.3124,B 9.7773,C 0.3347,E1 9.8406,E2 518.4013} C_DIS
LIN {X 50.2131,Y -126.8357,Z 169,A -65.9437,B 9.7775,C 0.3303,E1 9.8442,E2 517.0147} C_DIS
LIN {X 53.5904,Y -125.4446,Z 169,A -64.5052,B 9.7775,C 0.3305,E1 9.8479,E2 515.5871} C_DIS
LIN {X 56.8773,Y -123.9881,Z 169,A -63.0556,B 9.7775,C 0.3299,E1 9.8515,E2 514.144} C_DIS
LIN {X 59.9755,Y -122.5195,Z 169,A -61.6838,B 9.7775,C 0.3295,E1 9.855,E2 512.7797} C_DIS
LIN {X 63.0543,Y -120.9637,Z 169,A -60.159,B 9.7776,C 0.3257,E1 9.8588,E2 511.2439} C_DIS
LIN {X 66.6549,Y -119.0194,Z 169,A -58.3707,B 9.7778,C 0.3215,E1 9.8632,E2 509.4453} C_DIS
LIN {X 70.2155,Y -116.9548,Z 169,A -56.7625,B 9.7778,C 0.3215,E1 9.867,E2 507.8509} C_DIS
LIN {X 73.1794,Y -115.1234,Z 169,A -55.2017,B 9.7779,C 0.3169,E1 9.8708,E2 506.2763} C_DIS
LIN {X 76.8284,Y -112.7211,Z 169,A -53.4355,B 9.7779,C 0.3153,E1 9.8748,E2 504.5172} C_DIS
LIN {X 79.8821,Y -110.5773,Z 169,A -51.8591,B 9.7781,C 0.3123,E1 9.8784,E2 502.9381} C_DIS
LIN {X 83.2205,Y -108.0879,Z 169,A -50.1488,B 9.7781,C 0.31,E1 9.8822,E2 501.2311} C_DIS
LIN {X 86.4764,Y -105.5003,Z 169,A -48.4033,B 9.7783,C 0.3066,E1 9.886,E2 499.484} C_DIS
LIN {X 89.8492,Y -102.6432,Z 169,A -46.6083,B 9.7783,C 0.3044,E1 9.8898,E2 497.6951} C_DIS
LIN {X 92.6419,Y -100.1305,Z 169,A -45.0192,B 9.7784,C 0.3009,E1 9.8931,E2 496.103} C_DIS
LIN {X 95.451,Y -97.4554,Z 169,A -43.3799,B 9.7785,C 0.2972,E1 9.8964,E2 494.4607} C_DIS
LIN {X 98.3134,Y -94.568,Z 169,A -41.7192,B 9.7786,C 0.2946,E1 9.8996,E2 492.8042} C_DIS
LIN {X 101.1676,Y -91.5074,Z 169,A -40.0093,B 9.7787,C 0.2919,E1 9.9028,E2 491.0985} C_DIS
LIN {X 103.6486,Y -88.6882,Z 169,A -38.4788,B 9.7787,C 0.2894,E1 9.9056,E2 489.5724} C_DIS
LIN {X 106.1765,Y -85.6446,Z 169,A -36.7712,B 9.7789,C 0.2844,E1 9.9087,E2 487.8571} C_DIS
LIN {X 108.6219,Y -82.5222,Z 169,A -35.1925,B 9.7789,C 0.2826,E1 9.9113,E2 486.2879} C_DIS
LIN {X 110.8419,Y -79.5145,Z 169,A -33.5648,B 9.7791,C 0.2774,E1 9.914,E2 484.6512} C_DIS
LIN {X 113.2115,Y -76.1038,Z 169,A -31.9212,B 9.7791,C 0.2755,E1 9.9166,E2 483.0185} C_DIS
LIN {X 115.2436,Y -72.9891,Z 169,A -30.3031,B 9.7793,C 0.2702,E1 9.919,E2 481.3916} C_DIS
LIN {X 117.5135,Y -69.2753,Z 169,A -28.4705,B 9.7794,C 0.2654,E1 9.9217,E2 479.5564} C_DIS
LIN {X 119.8556,Y -65.1392,Z 169,A -26.5356,B 9.7795,C 0.2617,E1 9.9243,E2 477.6272} C_DIS
LIN {X 121.4395,Y -62.1324,Z 169,A -25.4174,B 9.7795,C 0.2655,E1 9.9257,E2 476.5465} C_DIS
LIN {X 122.7158,Y -59.5774,Z 169,A -24.0203,B 9.7797,C 0.2575,E1 9.9274,E2 475.1232} C_DIS
LIN {X 124.1736,Y -56.4762,Z 169,A -22.4741,B 9.7798,C 0.251,E1 9.9293,E2 473.5619} C_DIS
LIN {X 125.716,Y -52.9488,Z 169,A -21.01,B 9.7798,C 0.2503,E1 9.9309,E2 472.1154} C_DIS
LIN {X 127.0283,Y -49.7177,Z 169,A -19.7623,B 9.7798,C 0.2516,E1 9.9321,E2 470.8935} C_DIS
LIN {X 128.0399,Y -47.0577,Z 169,A -18.3903,B 9.78,C 0.244,E1 9.9335,E2 469.4981} C_DIS
LIN {X 129.2961,Y -43.4812,Z 169,A -16.8231,B 9.78,C 0.2402,E1 9.9349,E2 467.9322} C_DIS
LIN {X 130.3211,Y -40.3052,Z 169,A -15.4437,B 9.7802,C 0.2368,E1 9.9361,E2 466.5542} C_DIS
LIN {X 131.1478,Y -37.5353,Z 169,A -14.1201,B 9.7803,C 0.2307,E1 9.9371,E2 465.2155} C_DIS
LIN {X 132.0171,Y -34.3528,Z 169,A -12.7619,B 9.7803,C 0.2274,E1 9.9381,E2 463.8593} C_DIS
LIN {X 132.8433,Y -31.0005,Z 169,A -11.4989,B 9.7803,C 0.2278,E1 9.9389,E2 462.6184} C_DIS
LIN {X 133.5937,Y -27.5837,Z 169,A -10.1659,B 9.7804,C 0.2269,E1 9.9397,E2 461.3011} C_DIS
LIN {X 134.2092,Y -24.4137,Z 169,A -8.6791,B 9.7806,C 0.2198,E1 9.9404,E2 459.7964} C_DIS
LIN {X 134.7459,Y -21.2534,Z 169,A -7.355,B 9.7806,C 0.2165,E1 9.941,E2 458.4737} C_DIS
LIN {X 135.2049,Y -18.1054,Z 169,A -6.0036,B 9.7807,C 0.2122,E1 9.9416,E2 457.119} C_DIS
LIN {X 135.5976,Y -14.8791,Z 169,A -4.7238,B 9.7807,C 0.2103,E1 9.942,E2 455.8485} C_DIS
LIN {X 135.8955,Y -11.8566,Z 169,A -3.591,B 9.7807,C 0.2101,E1 9.9423,E2 454.7325} C_DIS
LIN {X 136.1057,Y -9.1586,Z 169,A -2.3264,B 9.7809,C 0.2037,E1 9.9425,E2 453.4507} C_DIS
LIN {X 136.2933,Y -5.6863,Z 169,A -1.0352,B 9.7809,C 0.2036,E1 9.9427,E2 452.1793} C_DIS
LIN {X 136.3878,Y -2.5502,Z 169,A 0.3851,B 9.781,C 0.1972,E1 9.9428,E2 450.7448} C_DIS
LIN {X 136.3986,Y 1.9023,Z 169,A 2.2484,B 9.7811,C 0.1919,E1 9.9428,E2 448.8805} C_DIS
LIN {X 136.3375,Y 4.5515,Z 169,A 3.4621,B 9.7813,C 0.1862,E1 9.9427,E2 447.6532} C_DIS
LIN {X 136.1761,Y 8.0151,Z 169,A 4.7839,B 9.7813,C 0.1853,E1 9.9425,E2 446.3469} C_DIS
LIN {X 135.943,Y 11.2946,Z 169,A 6.0265,B 9.7813,C 0.1846,E1 9.9422,E2 445.1203} C_DIS
LIN {X 135.6688,Y 14.2173,Z 169,A 7.2144,B 9.7813,C 0.1822,E1 9.9419,E2 443.9371} C_DIS
LIN {X 135.3574,Y 16.9411,Z 169,A 8.4998,B 9.7815,C 0.1756,E1 9.9415,E2 442.6339} C_DIS
LIN {X 134.9269,Y 20.0839,Z 169,A 9.8147,B 9.7815,C 0.1722,E1 9.941,E2 441.3199} C_DIS
LIN {X 134.3191,Y 23.7996,Z 169,A 11.3354,B 9.7815,C 0.1691,E1 9.9402,E2 439.8054} C_DIS
LIN {X 133.8206,Y 26.4688,Z 169,A 12.6043,B 9.7817,C 0.1628,E1 9.9396,E2 438.5195} C_DIS
LIN {X 133.0737,Y 29.992,Z 169,A 13.9819,B 9.7817,C 0.1617,E1 9.9387,E2 437.1575} C_DIS
LIN {X 132.304,Y 33.2225,Z 169,A 15.3572,B 9.7817,C 0.1583,E1 9.9378,E2 435.7834} C_DIS
LIN {X 131.4779,Y 36.355,Z 169,A 16.736,B 9.7818,C 0.154,E1 9.9368,E2 434.4013} C_DIS
LIN {X 130.6821,Y 39.1259,Z 169,A 17.9092,B 9.7818,C 0.1516,E1 9.9359,E2 433.2319} C_DIS
LIN {X 129.6881,Y 42.3041,Z 169,A 19.416,B 9.7819,C 0.1451,E1 9.9346,E2 431.7104} C_DIS
LIN {X 128.463,Y 45.8841,Z 169,A 20.8587,B 9.7819,C 0.1443,E1 9.9333,E2 430.2849} C_DIS
LIN {X 127.2901,Y 49.044,Z 169,A 22.0953,B 9.7819,C 0.1448,E1 9.9321,E2 429.0696} C_DIS
LIN {X 126.2019,Y 51.7854,Z 169,A 23.4793,B 9.782,C 0.138,E1 9.9306,E2 427.6666} C_DIS
LIN {X 124.6879,Y 55.3263,Z 169,A 25.0747,B 9.7821,C 0.1342,E1 9.9289,E2 426.0728} C_DIS
LIN {X 123.25,Y 58.4592,Z 169,A 26.4973,B 9.7821,C 0.131,E1 9.9272,E2 424.6523} C_DIS
LIN {X 121.7424,Y 61.5374,Z 169,A 27.8884,B 9.7821,C 0.1285,E1 9.9254,E2 423.2663} C_DIS
LIN {X 119.9973,Y 64.8786,Z 169,A 29.5542,B 9.7823,C 0.1225,E1 9.9233,E2 421.5893} C_DIS
LIN {X 117.8399,Y 68.7197,Z 169,A 31.3196,B 9.7823,C 0.1199,E1 9.9208,E2 419.8333} C_DIS
LIN {X 116.0493,Y 71.7022,Z 169,A 32.881,B 9.7823,C 0.1139,E1 9.9185,E2 418.2586} C_DIS
LIN {X 113.6316,Y 75.4746,Z 169,A 34.6484,B 9.7823,C 0.1121,E1 9.9158,E2 416.5044} C_DIS
LIN {X 111.595,Y 78.4541,Z 169,A 36.2181,B 9.7824,C 0.1072,E1 9.9133,E2 414.9272} C_DIS
LIN {X 109.0145,Y 82.002,Z 169,A 38.0208,B 9.7824,C 0.1039,E1 9.9103,E2 413.1286} C_DIS
LIN {X 106.4577,Y 85.2959,Z 169,A 39.7352,B 9.7824,C 0.1008,E1 9.9074,E2 411.4179} C_DIS
LIN {X 103.6853,Y 88.6451,Z 169,A 41.5416,B 9.7825,C 0.0973,E1 9.9041,E2 409.6132} C_DIS
LIN {X 101.1676,Y 91.5074,Z 169,A 43.1422,B 9.7825,C 0.0938,E1 9.9012,E2 408.012} C_DIS
LIN {X 98.3134,Y 94.568,Z 169,A 44.9089,B 9.7826,C 0.09,E1 9.8978,E2 406.2435} C_DIS
LIN {X 95.2,Y 97.7015,Z 169,A 46.6936,B 9.7826,C 0.0879,E1 9.8942,E2 404.4669} C_DIS
LIN {X 92.4741,Y 100.2847,Z 169,A 48.3005,B 9.7826,C 0.0841,E1 9.8909,E2 402.8559} C_DIS
LIN {X 89.1011,Y 103.293,Z 169,A 50.165,B 9.7826,C 0.0813,E1 9.887,E2 400.9949} C_DIS
LIN {X 85.5511,Y 106.2519,Z 169,A 52.046,B 9.7826,C 0.0792,E1 9.883,E2 399.1209} C_DIS
LIN {X 82.0552,Y 108.9744,Z 169,A 53.8838,B 9.7827,C 0.0765,E1 9.8789,E2 397.2856} C_DIS
LIN {X 78.9854,Y 111.2203,Z 169,A 55.5234,B 9.7827,C 0.0728,E1 9.8752,E2 395.6405} C_DIS
LIN {X 75.3766,Y 113.697,Z 169,A 57.3058,B 9.7827,C 0.0712,E1 9.8711,E2 393.8648} C_DIS
LIN {X 71.962,Y 115.8876,Z 169,A 58.9807,B 9.7827,C 0.0692,E1 9.8671,E2 392.1932} C_DIS
LIN {X 68.1924,Y 118.1451,Z 169,A 60.8034,B 9.7827,C 0.0671,E1 9.8627,E2 390.3732} C_DIS
LIN {X 64.3785,Y 120.266,Z 169,A 62.7456,B 9.7828,C 0.0621,E1 9.858,E2 388.4174} C_DIS
LIN {X 61.119,Y 121.9553,Z 169,A 64.119,B 9.7828,C 0.0639,E1 9.8546,E2 387.0648} C_DIS
LIN {X 58.0297,Y 123.4552,Z 169,A 65.551,B 9.7828,C 0.0624,E1 9.851,E2 385.634} C_DIS
LIN {X 54.5137,Y 125.0454,Z 169,A 67.1735,B 9.7828,C 0.0605,E1 9.8468,E2 384.0114} C_DIS
LIN {X 51.3795,Y 126.3655,Z 169,A 68.4168,B 9.7828,C 0.063,E1 9.8437,E2 382.7908} C_DIS
LIN {X 48.637,Y 127.4483,Z 169,A 69.8099,B 9.7828,C 0.0584,E1 9.84,E2 381.3789} C_DIS
LIN {X 45.214,Y 128.701,Z 169,A 71.3895,B 9.7828,C 0.0558,E1 9.8358,E2 379.7935} C_DIS
LIN {X 41.8153,Y 129.8442,Z 169,A 72.8057,B 9.7828,C 0.0565,E1 9.8321,E2 378.3885} C_DIS
LIN {X 38.7152,Y 130.8023,Z 169,A 74.2312,B 9.7828,C 0.054,E1 9.8283,E2 376.9555} C_DIS
LIN {X 35.9441,Y 131.5928,Z 169,A 75.4854,B 9.7828,C 0.0522,E1 9.8249,E2 375.6962} C_DIS
LIN {X 32.351,Y 132.52,Z 169,A 76.7817,B 9.7828,C 0.0568,E1 9.8215,E2 374.4324} C_DIS
LIN {X 29.5816,Y 133.1674,Z 169,A 78.2513,B 9.7828,C 0.0501,E1 9.8174,E2 372.9294} C_DIS
LIN {X 26.0806,Y 133.8955,Z 169,A 79.6463,B 9.7828,C 0.0516,E1 9.8136,E2 371.5478} C_DIS
LIN {X 22.8321,Y 134.4873,Z 169,A 81.0035,B 9.7828,C 0.0516,E1 9.8099,E2 370.1947} C_DIS
LIN {X 19.6777,Y 134.985,Z 169,A 82.34,B 9.7828,C 0.0512,E1 9.8062,E2 368.8592} C_DIS
LIN {X 16.463,Y 135.4145,Z 169,A 83.5188,B 9.7828,C 0.0546,E1 9.803,E2 367.7033} C_DIS
LIN {X 13.4122,Y 135.7508,Z 169,A 84.9823,B 9.7828,C 0.0505,E1 9.7989,E2 366.2189} C_DIS
LIN {X 10.0338,Y 136.0418,Z 169,A 86.3982,B 9.7828,C 0.0505,E1 9.7949,E2 364.8046} C_DIS
LIN {X 5.6863,Y 136.2933,Z 169,A 88.0804,B 9.7828,C 0.0533,E1 9.7903,E2 363.1411} C_DIS
LIN {X 3.0278,Y 136.3799,Z 169,A 89.458,B 9.7828,C 0.0478,E1 9.7864,E2 361.7322} C_DIS
LIN {X 0,Y 136.4135,Z 169,A 90.7296,B 9.7828,C 0.0478,E1 9.7828,E2 360.4613} C_DIS
LIN {X -3.7474,Y 136.3599,Z 169,A 92.2244,B 9.7828,C 0.0496,E1 9.7787,E2 358.9767} C_DIS
LIN {X -7.6171,Y 136.2007,Z 169,A 93.9419,B 9.7828,C 0.0481,E1 9.7738,E2 357.2491} C_DIS
LIN {X -10.7054,Y 135.9928,Z 169,A 95.1266,B 9.7828,C 0.0508,E1 9.7706,E2 356.0792} C_DIS
LIN {X -14.2173,Y 135.6688,Z 169,A 96.4613,B 9.7828,C 0.0542,E1 9.7669,E2 354.7632} C_DIS
LIN {X -17.3632,Y 135.3021,Z 169,A 97.9763,B 9.7828,C 0.051,E1 9.7627,E2 353.2263} C_DIS
LIN {X -21.6604,Y 134.6828,Z 169,A 99.7802,B 9.7828,C 0.0522,E1 9.7577,E2 351.426} C_DIS
LIN {X -25.2313,Y 134.0579,Z 169,A 101.153,B 9.7828,C 0.0561,E1 9.754,E2 350.0724} C_DIS
LIN {X -28.4035,Y 133.4218,Z 169,A 102.6976,B 9.7828,C 0.0532,E1 9.7497,E2 348.506} C_DIS
LIN {X -31.4875,Y 132.7281,Z 169,A 104.0376,B 9.7828,C 0.0538,E1 9.746,E2 347.1654} C_DIS
LIN {X -34.7637,Y 131.9076,Z 169,A 105.4366,B 9.7828,C 0.0553,E1 9.7423,E2 345.7697} C_DIS
LIN {X -37.5353,Y 131.1478,Z 169,A 106.7658,B 9.7828,C 0.0539,E1 9.7387,E2 344.4266} C_DIS
LIN {X -41.198,Y 130.0414,Z 169,A 108.2878,B 9.7828,C 0.057,E1 9.7346,E2 342.9161} C_DIS
LIN {X -44.3,Y 129.0179,Z 169,A 109.6483,B 9.7828,C 0.0586,E1 9.731,E2 341.558} C_DIS
LIN {X -47.4655,Y 127.8871,Z 169,A 111.0693,B 9.7828,C 0.0598,E1 9.7273,E2 340.1369} C_DIS
LIN {X -50.2131,Y 126.8357,Z 169,A 112.3133,B 9.7828,C 0.061,E1 9.7241,E2 338.8929} C_DIS
LIN {X -53.3537,Y 125.5469,Z 169,A 113.8959,B 9.7828,C 0.0596,E1 9.7199,E2 337.2924} C_DIS
LIN {X -56.8773,Y 123.9881,Z 169,A 115.3802,B 9.7828,C 0.0642,E1 9.7162,E2 335.8256} C_DIS
LIN {X -59.9755,Y 122.5195,Z 169,A 116.664,B 9.7828,C 0.0691,E1 9.713,E2 334.5621} C_DIS
LIN {X -62.654,Y 121.1739,Z 169,A 118.2441,B 9.7828,C 0.0646,E1 9.709,E2 332.9439} C_DIS
LIN {X -66.6549,Y 119.0194,Z 169,A 120.1354,B 9.7828,C 0.0677,E1 9.7044,E2 331.0564} C_DIS
LIN {X -70.2155,Y 116.9548,Z 169,A 121.7693,B 9.7828,C 0.0721,E1 9.7005,E2 329.4357} C_DIS
LIN {X -73.6011,Y 114.8535,Z 169,A 123.5117,B 9.7828,C 0.0735,E1 9.6964,E2 327.6863} C_DIS
LIN {X -77.0147,Y 112.5932,Z 169,A 125.1939,B 9.7828,C 0.077,E1 9.6925,E2 326.0103} C_DIS
LIN {X -79.8821,Y 110.5773,Z 169,A 126.7605,B 9.7828,C 0.0778,E1 9.6889,E2 324.4335} C_DIS
LIN {X -83.2205,Y 108.0879,Z 169,A 128.5037,B 9.7827,C 0.081,E1 9.685,E2 322.6927} C_DIS
LIN {X -86.1572,Y 105.7612,Z 169,A 130.1169,B 9.7827,C 0.0832,E1 9.6815,E2 321.0762} C_DIS
LIN {X -89.3563,Y 103.0733,Z 169,A 131.8669,B 9.7827,C 0.0867,E1 9.6778,E2 319.3285} C_DIS
LIN {X -92.4741,Y 100.2847,Z 169,A 133.6144,B 9.7826,C 0.0904,E1 9.6742,E2 317.5839} C_DIS
LIN {X -95.365,Y 97.5397,Z 169,A 135.2781,B 9.7826,C 0.094,E1 9.6708,E2 315.9232} C_DIS
LIN {X -98.1549,Y 94.7318,Z 169,A 136.9882,B 9.7826,C 0.0966,E1 9.6675,E2 314.2089} C_DIS
LIN {X -100.7277,Y 91.9922,Z 169,A 138.5559,B 9.7826,C 0.1003,E1 9.6645,E2 312.6442} C_DIS
LIN {X -103.0733,Y 89.3563,Z 169,A 140.1124,B 9.7825,C 0.1022,E1 9.6616,E2 311.0802} C_DIS
LIN {X -105.7612,Y 86.1572,Z 169,A 141.8599,B 9.7825,C 0.1063,E1 9.6585,E2 309.3353} C_DIS
LIN {X -108.0879,Y 83.2205,Z 169,A 143.4807,B 9.7825,C 0.1091,E1 9.6558,E2 307.7104} C_DIS
LIN {X -110.5773,Y 79.8821,Z 169,A 145.2229,B 9.7824,C 0.1134,E1 9.6529,E2 305.9709} C_DIS
LIN {X -112.7211,Y 76.8284,Z 169,A 146.9047,B 9.7824,C 0.1151,E1 9.6502,E2 304.2766} C_DIS
LIN {X -115.1234,Y 73.1794,Z 169,A 148.6387,B 9.7823,C 0.1215,E1 9.6476,E2 302.557} C_DIS
LIN {X -117.0697,Y 70.0227,Z 169,A 150.216,B 9.7823,C 0.125,E1 9.6453,E2 300.9789} C_DIS
LIN {X -119.129,Y 66.4599,Z 169,A 152.0998,B 9.7823,C 0.1267,E1 9.6427,E2 299.078} C_DIS
LIN {X -121.3757,Y 62.2577,Z 169,A 153.8255,B 9.7821,C 0.1369,E1 9.6405,E2 297.3881} C_DIS
LIN {X -122.7158,Y 59.5774,Z 169,A 155.2695,B 9.7821,C 0.1369,E1 9.6387,E2 295.9229} C_DIS
LIN {X -124.1736,Y 56.4762,Z 169,A 156.8603,B 9.7821,C 0.1379,E1 9.6368,E2 294.315} C_DIS
LIN {X -125.7449,Y 52.8796,Z 169,A 158.4119,B 9.782,C 0.1441,E1 9.6351,E2 292.7769} C_DIS
LIN {X -126.8357,Y 50.2131,Z 169,A 159.6244,B 9.782,C 0.1474,E1 9.6338,E2 291.5655} C_DIS
LIN {X -128.0622,Y 46.9958,Z 169,A 161.065,B 9.7819,C 0.1515,E1 9.6324,E2 290.1271} C_DIS
LIN {X -129.2961,Y 43.4812,Z 169,A 162.6756,B 9.7818,C 0.155,E1 9.631,E2 288.5125} C_DIS
LIN {X -130.3211,Y 40.3052,Z 169,A 164.096,B 9.7818,C 0.1586,E1 9.6298,E2 287.0913} C_DIS
LIN {X -131.1478,Y 37.5353,Z 169,A 165.3273,B 9.7817,C 0.1617,E1 9.6288,E2 285.8592} C_DIS
LIN {X -132.0171,Y 34.3528,Z 169,A 166.8591,B 9.7817,C 0.163,E1 9.6277,E2 284.3109} C_DIS
LIN {X -132.8044,Y 31.1712,Z 169,A 168.1272,B 9.7816,C 0.1689,E1 9.6269,E2 283.0576} C_DIS
LIN {X -133.6212,Y 27.4485,Z 169,A 169.7805,B 9.7816,C 0.1725,E1 9.6259,E2 281.3994} C_DIS
LIN {X -134.2291,Y 24.3026,Z 169,A 171.1202,B 9.7814,C 0.1765,E1 9.6252,E2 280.0619} C_DIS
LIN {X -134.7459,Y 21.2534,Z 169,A 172.4305,B 9.7814,C 0.18,E1 9.6246,E2 278.7516} C_DIS
LIN {X -135.2049,Y 18.1054,Z 169,A 173.7848,B 9.7814,C 0.1836,E1 9.6241,E2 277.3964} C_DIS
LIN {X -135.6153,Y 14.715,Z 169,A 175.1709,B 9.7812,C 0.1886,E1 9.6237,E2 276.0176} C_DIS
LIN {X -135.8955,Y 11.8566,Z 169,A 176.31,B 9.7812,C 0.1933,E1 9.6234,E2 274.8881} C_DIS
LIN {X -136.1057,Y 9.1586,Z 169,A 177.7587,B 9.7812,C 0.1911,E1 9.6231,E2 273.4021} C_DIS
LIN {X -136.3048,Y 5.3895,Z 169,A 179.2133,B 9.781,C 0.198,E1 9.6229,E2 271.9652} C_DIS
LIN {X -136.3903,Y 2.4025,Z 169,A -179.5476,B 9.781,C 0.2019,E1 9.6229,E2 270.7293} C_DIS
LIN {X -136.3986,Y -1.9023,Z 169,A -177.669,B 9.7809,C 0.206,E1 9.6229,E2 268.8437} C_DIS
LIN {X -136.3375,Y -4.5515,Z 169,A -176.4163,B 9.7809,C 0.2067,E1 9.6229,E2 267.5749} C_DIS
LIN {X -136.1761,Y -8.0151,Z 169,A -175.055,B 9.7807,C 0.2126,E1 9.6232,E2 266.2267} C_DIS
LIN {X -135.9745,Y -10.9216,Z 169,A -173.743,B 9.7807,C 0.2146,E1 9.6234,E2 264.9049} C_DIS
LIN {X -135.6688,Y -14.2173,Z 169,A -172.3477,B 9.7806,C 0.2185,E1 9.6238,E2 263.5102} C_DIS
LIN {X -135.2768,Y -17.5567,Z 169,A -170.994,B 9.7805,C 0.2236,E1 9.6243,E2 262.165} C_DIS
LIN {X -134.6828,Y -21.6604,Z 169,A -169.1882,B 9.7804,C 0.2275,E1 9.625,E2 260.3528} C_DIS
LIN {X -134.0579,Y -25.2313,Z 169,A -167.6187,B 9.7804,C 0.231,E1 9.6258,E2 258.7788} C_DIS
LIN {X -133.4218,Y -28.4035,Z 169,A -166.258,B 9.7802,C 0.2348,E1 9.6266,E2 257.419} C_DIS
LIN {X -132.7446,Y -31.419,Z 169,A -164.8898,B 9.7802,C 0.2372,E1 9.6275,E2 256.0432} C_DIS
LIN {X -131.9076,Y -34.7637,Z 169,A -163.4664,B 9.7801,C 0.2417,E1 9.6285,E2 254.6241} C_DIS
LIN {X -131.1478,Y -37.5353,Z 169,A -162.1301,B 9.7801,C 0.2427,E1 9.6295,E2 253.2727} C_DIS
LIN {X -130.1955,Y -40.7157,Z 169,A -160.7504,B 9.7799,C 0.2468,E1 9.6306,E2 251.896} C_DIS
LIN {X -129.0179,Y -44.3,Z 169,A -159.2131,B 9.7798,C 0.252,E1 9.632,E2 250.3657} C_DIS
LIN {X -127.8871,Y -47.4655,Z 169,A -157.7794,B 9.7798,C 0.2554,E1 9.6333,E2 248.9304} C_DIS
LIN {X -126.8357,Y -50.2131,Z 169,A -156.3758,B 9.7798,C 0.2557,E1 9.6348,E2 247.5068} C_DIS
LIN {X -125.5469,Y -53.3537,Z 169,A -154.9444,B 9.7796,C 0.2593,E1 9.6364,E2 246.0758} C_DIS
LIN {X -123.9881,Y -56.8773,Z 169,A -153.4346,B 9.7794,C 0.2656,E1 9.6381,E2 244.5806} C_DIS
LIN {X -122.5195,Y -59.9755,Z 169,A -151.9727,B 9.7794,C 0.2689,E1 9.6398,E2 243.117} C_DIS
LIN {X -121.1739,Y -62.654,Z 169,A -150.5866,B 9.7794,C 0.2698,E1 9.6416,E2 241.7158} C_DIS
LIN {X -119.129,Y -66.4599,Z 169,A -148.7225,B 9.7792,C 0.2734,E1 9.6441,E2 239.8466} C_DIS
LIN {X -116.9548,Y -70.2155,Z 169,A -146.9632,B 9.7791,C 0.279,E1 9.6466,E2 238.0964} C_DIS
LIN {X -114.7744,Y -73.7246,Z 169,A -145.1639,B 9.779,C 0.282,E1 9.6493,E2 236.2901} C_DIS
LIN {X -112.5932,Y -77.0147,Z 169,A -143.4662,B 9.7789,C 0.2852,E1 9.652,E2 234.5883} C_DIS
LIN {X -110.0612,Y -80.5917,Z 169,A -141.7053,B 9.7787,C 0.2909,E1 9.6548,E2 232.8384} C_DIS
LIN {X -107.6883,Y -83.736,Z 169,A -140.0017,B 9.7787,C 0.2937,E1 9.6577,E2 231.1294} C_DIS
LIN {X -105.1282,Y -86.9282,Z 169,A -138.2051,B 9.7786,C 0.296,E1 9.6609,E2 229.3238} C_DIS
LIN {X -102.3426,Y -90.1913,Z 169,A -136.3681,B 9.7785,C 0.2992,E1 9.6643,E2 227.4831} C_DIS
LIN {X -99.3115,Y -93.5184,Z 169,A -134.4648,B 9.7784,C 0.3028,E1 9.6679,E2 225.579} C_DIS
LIN {X -96.2218,Y -96.6945,Z 169,A -132.5876,B 9.7783,C 0.3062,E1 9.6716,E2 223.7004} C_DIS
LIN {X -92.9137,Y -99.8774,Z 169,A -130.6647,B 9.7781,C 0.31,E1 9.6755,E2 221.7788} C_DIS
LIN {X -89.8492,Y -102.6432,Z 169,A -128.8737,B 9.7781,C 0.3121,E1 9.6793,E2 219.9812} C_DIS
LIN {X -86.6631,Y -105.3478,Z 169,A -127.2064,B 9.7779,C 0.317,E1 9.6828,E2 218.3255} C_DIS
LIN {X -83.5144,Y -107.8601,Z 169,A -125.4464,B 9.7779,C 0.3185,E1 9.6867,E2 216.5572} C_DIS
LIN {X -80.4091,Y -110.1954,Z 169,A -123.8541,B 9.7778,C 0.322,E1 9.6902,E2 214.9703} C_DIS
LIN {X -77.5502,Y -112.2257,Z 169,A -122.3698,B 9.7777,C 0.3241,E1 9.6936,E2 213.4848} C_DIS
LIN {X -74.478,Y -114.287,Z 169,A -120.7988,B 9.7777,C 0.3261,E1 9.6973,E2 211.9118} C_DIS
LIN {X -71.1516,Y -116.387,Z 169,A -119.0564,B 9.7777,C 0.3267,E1 9.7015,E2 210.1582} C_DIS
LIN {X -67.2152,Y -118.7045,Z 169,A -117.0777,B 9.7776,C 0.3281,E1 9.7063,E2 208.1721} C_DIS
LIN {X -63.7874,Y -120.5787,Z 169,A -115.5593,B 9.7774,C 0.3326,E1 9.71,E2 206.6692} C_DIS
LIN {X -61.119,Y -121.9553,Z 169,A -114.2911,B 9.7774,C 0.334,E1 9.7131,E2 205.4002} C_DIS
LIN {X -58.0297,Y -123.4552,Z 169,A -112.7761,B 9.7774,C 0.3342,E1 9.717,E2 203.8759} C_DIS
LIN {X -54.4545,Y -125.071,Z 169,A -111.2038,B 9.7772,C 0.3375,E1 9.721,E2 202.3131} C_DIS
LIN {X -51.3795,Y -126.3655,Z 169,A -109.9192,B 9.7772,C 0.3413,E1 9.7242,E2 201.0432} C_DIS
LIN {X -48.213,Y -127.6071,Z 169,A -108.3432,B 9.7772,C 0.3396,E1 9.7284,E2 199.4485} C_DIS
LIN {X -44.9147,Y -128.8048,Z 169,A -106.9091,B 9.7772,C 0.3417,E1 9.7322,E2 198.0192} C_DIS
LIN {X -41.894,Y -129.8191,Z 169,A -105.5241,B 9.7771,C 0.3417,E1 9.7358,E2 196.6281} C_DIS
LIN {X -38.7152,Y -130.8023,Z 169,A -104.0781,B 9.7771,C 0.3418,E1 9.7397,E2 195.1757} C_DIS
LIN {X -35.9441,Y -131.5928,Z 169,A -102.9098,B 9.7771,C 0.3435,E1 9.7429,E2 194.0125} C_DIS
LIN {X -32.351,Y -132.52,Z 169,A -101.5061,B 9.7769,C 0.3476,E1 9.7466,E2 192.6281} C_DIS
LIN {X -29.5816,Y -133.1674,Z 169,A -100.0285,B 9.7771,C 0.3424,E1 9.7507,E2 191.1143} C_DIS
LIN {X -26.0285,Y -133.9055,Z 169,A -98.5846,B 9.777,C 0.3447,E1 9.7547,E2 189.6802} C_DIS
LIN {X -22.8321,Y -134.4873,Z 169,A -97.2626,B 9.777,C 0.3461,E1 9.7583,E2 188.3632} C_DIS
LIN {X -19.4532,Y -135.0171,Z 169,A -95.885,B 9.7769,C 0.3478,E1 9.7621,E2 186.9926} C_DIS
LIN {X -16.5369,Y -135.4057,Z 169,A -94.7416,B 9.7769,C 0.3501,E1 9.7652,E2 185.8606} C_DIS
LIN {X -13.4122,Y -135.7508,Z 169,A -93.2716,B 9.7769,C 0.3472,E1 9.7693,E2 184.3711} C_DIS
LIN {X -10.7054,Y -135.9928,Z 169,A -92.1309,B 9.7769,C 0.3473,E1 9.7725,E2 183.2301} C_DIS
LIN {X -7.6171,Y -136.2007,Z 169,A -90.7161,B 9.7769,C 0.3449,E1 9.7765,E2 181.8001} C_DIS
LIN {X -4.5515,Y -136.3375,Z 169,A -89.5467,B 9.7769,C 0.3475,E1 9.7797,E2 180.6453} C_DIS
LIN {X -1.1206,Y -136.4073,Z 169,A -88.2533,B 9.7768,C 0.3505,E1 9.7833,E2 179.3701} C_DIS
LIN {X 0.9918,Y -136.4057,Z 169,A -87.4754,B 9.7768,C 0.3528,E1 9.7854,E2 178.6056} C_DIS
Enddeposition()
LIN {X 0.9918,Y -136.4057,Z 169,A -87.4754,B 9.7768,C 0.3528,E1 9.7854,E2 178.6056} C_DIS
Startdeposition()
$VEL.CP = VEL_PRINT
LIN {X -0.3765,Y -137.3238,Z 169,A -88.4276,B 9.7415,C 0.3679,E1 9.7479,E2 179.651} C_DIS
LIN {X -4.5431,Y -137.2505,Z 169,A -90.2008,B 9.7415,C 0.3688,E1 9.7429,E2 181.4294} C_DIS
LIN {X -11.3466,Y -136.8542,Z 169,A -92.7313,B 9.7417,C 0.3619,E1 9.736,E2 183.9213} C_DIS
LIN {X -13.6065,Y -136.6487,Z 169,A -94.2235,B 9.7413,C 0.3733,E1 9.7316,E2 185.4829} C_DIS
LIN {X -17.1928,Y -136.2446,Z 169,A -95.5358,B 9.7415,C 0.3689,E1 9.728,E2 186.7715} C_DIS
LIN {X -20.8639,Y -135.7294,Z 169,A -97.3123,B 9.7413,C 0.3732,E1 9.7231,E2 188.5773} C_DIS
LIN {X -24.5731,Y -135.1075,Z 169,A -98.4103,B 9.7417,C 0.3628,E1 9.7202,E2 189.6163} C_DIS
LIN {X -27.4486,Y -134.5523,Z 169,A -99.8195,B 9.7416,C 0.3661,E1 9.7163,E2 191.0496} C_DIS
LIN {X -31.813,Y -133.5881,Z 169,A -102.0293,B 9.7413,C 0.3723,E1 9.7101,E2 193.3033} C_DIS
LIN {X -35.6691,Y -132.6104,Z 169,A -103.2286,B 9.7417,C 0.3618,E1 9.7071,E2 194.4449} C_DIS
LIN {X -39.0274,Y -131.6616,Z 169,A -104.6846,B 9.7417,C 0.3608,E1 9.7032,E2 195.9012} C_DIS
LIN {X -41.9016,Y -130.7744,Z 169,A -105.9857,B 9.7417,C 0.3608,E1 9.6997,E2 197.2083} C_DIS
LIN {X -45.2191,Y -129.6648,Z 169,A -107.4631,B 9.7418,C 0.3599,E1 9.6958,E2 198.6882} C_DIS
LIN {X -48.3988,Y -128.5118,Z 169,A -108.8917,B 9.7418,C 0.359,E1 9.692,E2 200.1191} C_DIS
LIN {X -51.7133,Y -127.2146,Z 169,A -110.3964,B 9.7418,C 0.358,E1 9.6881,E2 201.6264} C_DIS
LIN {X -54.7239,Y -125.9484,Z 169,A -111.733,B 9.7419,C 0.356,E1 9.6847,E2 202.9598} C_DIS
LIN {X -58.4404,Y -124.2701,Z 169,A -113.4428,B 9.742,C 0.3543,E1 9.6803,E2 204.6707} C_DIS
LIN {X -61.5558,Y -122.7566,Z 169,A -114.891,B 9.742,C 0.3527,E1 9.6767,E2 206.1194} C_DIS
LIN {X -64.0278,Y -121.483,Z 169,A -116.2676,B 9.742,C 0.3555,E1 9.6732,E2 207.523} C_DIS
LIN {X -67.8918,Y -119.3689,Z 169,A -118.0286,B 9.7421,C 0.3516,E1 9.669,E2 209.2744} C_DIS
LIN {X -71.9466,Y -116.9697,Z 169,A -120.2495,B 9.7421,C 0.3539,E1 9.6636,E2 211.5271} C_DIS
LIN {X -74.9683,Y -115.0565,Z 169,A -121.4318,B 9.7423,C 0.3456,E1 9.6609,E2 212.6704} C_DIS
LIN {X -78.2541,Y -112.8474,Z 169,A -123.1395,B 9.7423,C 0.3441,E1 9.6569,E2 214.3848} C_DIS
LIN {X -81.5675,Y -110.4764,Z 169,A -124.9095,B 9.7424,C 0.3427,E1 9.6529,E2 216.1632} C_DIS
LIN {X -84.411,Y -108.3195,Z 169,A -126.3914,B 9.7425,C 0.3401,E1 9.6497,E2 217.6439} C_DIS
LIN {X -87.9409,Y -105.474,Z 169,A -128.2323,B 9.7427,C 0.3358,E1 9.6457,E2 219.478} C_DIS
LIN {X -91.0567,Y -102.7954,Z 169,A -130.0076,B 9.7427,C 0.3338,E1 9.6419,E2 221.2604} C_DIS
LIN {X -94.432,Y -99.7039,Z 169,A -131.9628,B 9.7428,C 0.331,E1 9.6379,E2 223.2207} C_DIS
LIN {X -97.6715,Y -96.5329,Z 169,A -133.8443,B 9.7429,C 0.3271,E1 9.6342,E2 225.1004} C_DIS
LIN {X -100.7093,Y -93.3592,Z 169,A -135.5294,B 9.7432,C 0.3206,E1 9.631,E2 226.7662} C_DIS
LIN {X -103.0427,Y -90.7769,Z 169,A -137.3521,B 9.743,C 0.3245,E1 9.6275,E2 228.6346} C_DIS
LIN {X -106.3239,Y -86.9104,Z 169,A -139.3281,B 9.7433,C 0.3173,E1 9.624,E2 230.5923} C_DIS
LIN {X -108.9905,Y -83.5421,Z 169,A -141.0981,B 9.7434,C 0.3129,E1 9.621,E2 232.3587} C_DIS
LIN {X -111.3572,Y -80.3608,Z 169,A -142.7166,B 9.7436,C 0.3084,E1 9.6183,E2 233.9718} C_DIS
LIN {X -113.5828,Y -77.1829,Z 169,A -144.4452,B 9.7436,C 0.3067,E1 9.6156,E2 235.7132} C_DIS
LIN {X -116.0116,Y -73.4817,Z 169,A -146.3326,B 9.7437,C 0.303,E1 9.6127,E2 237.6047} C_DIS
LIN {X -118.3683,Y -69.6215,Z 169,A -148.2585,B 9.7438,C 0.2991,E1 9.6099,E2 239.5342} C_DIS
LIN {X -120.6835,Y -65.5267,Z 169,A -150.3632,B 9.7439,C 0.2968,E1 9.6071,E2 241.6554} C_DIS
LIN {X -122.4934,Y -62.0731,Z 169,A -151.7821,B 9.7441,C 0.2888,E1 9.6053,E2 243.0473} C_DIS
LIN {X -124.0631,Y -58.8739,Z 169,A -153.3495,B 9.7442,C 0.2865,E1 9.6034,E2 244.6237} C_DIS
LIN {X -125.5836,Y -55.5583,Z 169,A -154.7999,B 9.7444,C 0.2812,E1 9.6017,E2 246.0642} C_DIS
LIN {X -126.8234,Y -52.6646,Z 169,A -156.1751,B 9.7444,C 0.2788,E1 9.6002,E2 247.4462} C_DIS
LIN {X -128.1022,Y -49.4731,Z 169,A -157.6491,B 9.7445,C 0.2757,E1 9.5987,E2 248.924} C_DIS
LIN {X -130.1247,Y -43.8806,Z 169,A -160.007,B 9.7448,C 0.2668,E1 9.5965,E2 251.2648} C_DIS
LIN {X -132.3556,Y -36.6038,Z 169,A -163.3355,B 9.7449,C 0.2608,E1 9.5938,E2 254.6098} C_DIS
LIN {X -133.1512,Y -33.5931,Z 169,A -164.6279,B 9.745,C 0.257,E1 9.5929,E2 255.9002} C_DIS
LIN {X -133.8768,Y -30.5732,Z 169,A -165.9976,B 9.745,C 0.2547,E1 9.5921,E2 257.278} C_DIS
LIN {X -134.6104,Y -27.1628,Z 169,A -167.5088,B 9.7452,C 0.2516,E1 9.5912,E2 258.7948} C_DIS
LIN {X -135.3153,Y -23.4122,Z 169,A -169.0631,B 9.7453,C 0.2463,E1 9.5904,E2 260.3432} C_DIS
LIN {X -135.8778,Y -19.8794,Z 169,A -170.6576,B 9.7453,C 0.2439,E1 9.5897,E2 261.949} C_DIS
LIN {X -136.3615,Y -16.2267,Z 169,A -172.1635,B 9.7455,C 0.2389,E1 9.5892,E2 263.4495} C_DIS
LIN {X -136.7298,Y -12.7622,Z 169,A -173.6389,B 9.7455,C 0.2351,E1 9.5888,E2 264.9263} C_DIS
LIN {X -137.0541,Y -8.6014,Z 169,A -175.4201,B 9.7457,C 0.2307,E1 9.5884,E2 266.7108} C_DIS
LIN {X -137.2403,Y -4.8145,Z 169,A -177.1166,B 9.7457,C 0.2282,E1 9.5882,E2 268.4199} C_DIS
LIN {X -137.3219,Y -0.8817,Z 169,A -178.6601,B 9.7459,C 0.2217,E1 9.5882,E2 269.9499} C_DIS
LIN {X -137.3114,Y 1.8864,Z 169,A -179.889,B 9.7459,C 0.2196,E1 9.5882,E2 271.1867} C_DIS
LIN {X -137.2064,Y 5.6845,Z 169,A 178.5185,B 9.746,C 0.2151,E1 9.5884,E2 272.7786} C_DIS
LIN {X -137.0386,Y 8.8526,Z 169,A 177.1885,B 9.7461,C 0.2114,E1 9.5886,E2 274.108} C_DIS
LIN {X -136.7764,Y 12.268,Z 169,A 175.6856,B 9.7461,C 0.2085,E1 9.5889,E2 275.6186} C_DIS
LIN {X -136.3226,Y 16.5527,Z 169,A 173.9253,B 9.7463,C 0.2026,E1 9.5895,E2 277.3724} C_DIS
LIN {X -135.7944,Y 20.4437,Z 169,A 172.1802,B 9.7463,C 0.1998,E1 9.5902,E2 279.129} C_DIS
LIN {X -135.1983,Y 24.0662,Z 169,A 170.694,B 9.7465,C 0.1946,E1 9.5909,E2 280.6079} C_DIS
LIN {X -134.5521,Y 27.4493,Z 169,A 169.2191,B 9.7465,C 0.1911,E1 9.5917,E2 282.086} C_DIS
LIN {X -133.7231,Y 31.2462,Z 169,A 167.6186,B 9.7466,C 0.1861,E1 9.5927,E2 283.6823} C_DIS
LIN {X -133.0008,Y 34.1859,Z 169,A 166.3309,B 9.7466,C 0.183,E1 9.5935,E2 284.9717} C_DIS
LIN {X -132.02,Y 37.8031,Z 169,A 164.7383,B 9.7468,C 0.1791,E1 9.5947,E2 286.5662} C_DIS
LIN {X -131.2123,Y 40.5111,Z 169,A 163.5182,B 9.7468,C 0.1765,E1 9.5957,E2 287.7901} C_DIS
LIN {X -129.8718,Y 44.6221,Z 169,A 161.0181,B 9.7467,C 0.1838,E1 9.5981,E2 290.373} C_DIS
LIN {X -128.0615,Y 49.5779,Z 169,A 159.3811,B 9.747,C 0.1678,E1 9.5996,E2 291.939} C_DIS
LIN {X -126.6558,Y 53.066,Z 169,A 157.8772,B 9.747,C 0.1623,E1 9.6012,E2 293.4333} C_DIS
LIN {X -125.3127,Y 56.164,Z 169,A 156.4039,B 9.747,C 0.1597,E1 9.6028,E2 294.913} C_DIS
LIN {X -123.6126,Y 59.8167,Z 169,A 154.4318,B 9.747,C 0.1605,E1 9.6053,E2 296.9188} C_DIS
LIN {X -122.1646,Y 62.719,Z 169,A 153.4975,B 9.7473,C 0.1494,E1 9.6064,E2 297.8005} C_DIS
LIN {X -117.2279,Y 71.5256,Z 169,A 149.1536,B 9.7473,C 0.1411,E1 9.6124,E2 302.1564} C_DIS
LIN {X -115.2579,Y 74.6581,Z 169,A 147.4882,B 9.7473,C 0.1394,E1 9.6149,E2 303.8351} C_DIS
LIN {X -112.9517,Y 78.1042,Z 169,A 145.5193,B 9.7473,C 0.1395,E1 9.618,E2 305.8311} C_DIS
LIN {X -107.5044,Y 85.4459,Z 169,A 142.2004,B 9.7476,C 0.1215,E1 9.6235,E2 309.0856} C_DIS
LIN {X -104.4251,Y 89.1834,Z 169,A 139.8033,B 9.7476,C 0.1238,E1 9.6278,E2 311.5267} C_DIS
LIN {X -101.4681,Y 92.534,Z 169,A 137.9825,B 9.7476,C 0.1189,E1 9.6312,E2 313.3403} C_DIS
LIN {X -98.8031,Y 95.3739,Z 169,A 136.3041,B 9.7476,C 0.1164,E1 9.6344,E2 315.0236} C_DIS
LIN {X -96.0381,Y 98.1575,Z 169,A 134.5995,B 9.7477,C 0.1142,E1 9.6378,E2 316.7348} C_DIS
LIN {X -92.7805,Y 101.2423,Z 169,A 132.9283,B 9.7478,C 0.1067,E1 9.6412,E2 318.3796} C_DIS
LIN {X -90.2747,Y 103.4827,Z 169,A 131.311,B 9.7478,C 0.108,E1 9.6446,E2 320.0218} C_DIS
LIN {X -87.0593,Y 106.2022,Z 169,A 129.5249,B 9.7478,C 0.1052,E1 9.6485,E2 321.8097} C_DIS
LIN {X -83.9069,Y 108.7101,Z 169,A 127.8769,B 9.7478,C 0.1015,E1 9.6521,E2 323.4522} C_DIS
LIN {X -81.1173,Y 110.8072,Z 169,A 125.9347,B 9.7478,C 0.108,E1 9.6566,E2 325.4518} C_DIS
LIN {X -77.5625,Y 113.3238,Z 169,A 124.7111,B 9.7479,C 0.0938,E1 9.6592,E2 326.6017} C_DIS
LIN {X -74.5952,Y 115.2987,Z 169,A 122.9745,B 9.7479,C 0.0961,E1 9.6633,E2 328.3674} C_DIS
LIN {X -70.6688,Y 117.7467,Z 169,A 121.0438,B 9.7479,C 0.0931,E1 9.6679,E2 330.2965} C_DIS
LIN {X -66.2493,Y 120.2885,Z 169,A 119.1595,B 9.748,C 0.0853,E1 9.6724,E2 332.1493} C_DIS
LIN {X -63.4905,Y 121.7652,Z 169,A 117.647,B 9.748,C 0.0875,E1 9.6762,E2 333.6859} C_DIS
LIN {X -58.847,Y 124.0759,Z 169,A 115.5294,B 9.748,C 0.0837,E1 9.6815,E2 335.796} C_DIS
LIN {X -55.4634,Y 125.6261,Z 169,A 113.9533,B 9.748,C 0.0823,E1 9.6855,E2 337.3737} C_DIS
LIN {X -52.7981,Y 126.7676,Z 169,A 112.6781,B 9.748,C 0.0821,E1 9.6888,E2 338.6558} C_DIS
LIN {X -49.6751,Y 128.0237,Z 169,A 111.2376,B 9.748,C 0.0813,E1 9.6926,E2 340.0995} C_DIS
LIN {X -43.8292,Y 130.1419,Z 169,A 108.8572,B 9.7481,C 0.0745,E1 9.6988,E2 342.452} C_DIS
LIN {X -41.2313,Y 130.9886,Z 169,A 107.4297,B 9.7481,C 0.0791,E1 9.7027,E2 343.9137} C_DIS
LIN {X -37.2033,Y 132.188,Z 169,A 105.7928,B 9.7481,C 0.0753,E1 9.707,E2 345.5352} C_DIS
LIN {X -33.4256,Y 133.1937,Z 169,A 104.0627,B 9.7481,C 0.076,E1 9.7117,E2 347.2762} C_DIS
LIN {X -29.2004,Y 134.1831,Z 169,A 102.3655,B 9.7481,C 0.0726,E1 9.7163,E2 348.9584} C_DIS
LIN {X -25.2371,Y 134.9857,Z 169,A 100.6841,B 9.7481,C 0.0714,E1 9.7209,E2 350.6381} C_DIS
LIN {X -22.6275,Y 135.4465,Z 169,A 99.4049,B 9.7481,C 0.0744,E1 9.7245,E2 351.9377} C_DIS
LIN {X -17.5995,Y 136.1913,Z 169,A 97.4064,B 9.7481,C 0.071,E1 9.73,E2 353.9201} C_DIS
LIN {X -13.5386,Y 136.6552,Z 169,A 95.6291,B 9.7481,C 0.0718,E1 9.7349,E2 355.7053} C_DIS
LIN {X -9.0205,Y 137.0283,Z 169,A 93.2824,B 9.7481,C 0.0807,E1 9.7416,E2 358.1061} C_DIS
LIN {X -4.4142,Y 137.2541,Z 169,A 91.9904,B 9.7481,C 0.0675,E1 9.745,E2 359.3205} C_DIS
LIN {X 0.4004,Y 137.3236,Z 169,A 89.7696,B 9.7481,C 0.0717,E1 9.7513,E2 361.5662} C_DIS
LIN {X 4.7143,Y 137.2439,Z 169,A 87.5319,B 9.7481,C 0.0809,E1 9.7577,E2 363.8561} C_DIS
LIN {X 9.4009,Y 137.0028,Z 169,A 86.2241,B 9.7481,C 0.0676,E1 9.7611,E2 365.0843} C_DIS
LIN {X 16.3191,Y 136.3505,Z 169,A 83.1907,B 9.7481,C 0.0712,E1 9.7696,E2 368.1331} C_DIS
LIN {X 21.2804,Y 135.6649,Z 169,A 81.1787,B 9.7481,C 0.0704,E1 9.7751,E2 370.135} C_DIS
LIN {X 24.6148,Y 135.1001,Z 169,A 79.7237,B 9.7481,C 0.072,E1 9.7791,E2 371.5949} C_DIS
LIN {X 27.9704,Y 134.4461,Z 169,A 78.2955,B 9.7481,C 0.0728,E1 9.783,E2 373.023} C_DIS
LIN {X 33.0699,Y 133.284,Z 169,A 76.1877,B 9.7481,C 0.0726,E1 9.7887,E2 375.1212} C_DIS
LIN {X 37.096,Y 132.218,Z 169,A 74.4199,B 9.7481,C 0.0745,E1 9.7935,E2 376.8923} C_DIS
LIN {X 40.2939,Y 131.2787,Z 169,A 73.0118,B 9.7481,C 0.076,E1 9.7973,E2 378.3023} C_DIS
LIN {X 43.6173,Y 130.2124,Z 169,A 71.5737,B 9.7481,C 0.0768,E1 9.8011,E2 379.738} C_DIS
LIN {X 46.821,Y 129.0951,Z 169,A 70.146,B 9.7481,C 0.0784,E1 9.8048,E2 381.167} C_DIS
LIN {X 50.2617,Y 127.7957,Z 169,A 68.6269,B 9.7481,C 0.0797,E1 9.8088,E2 382.6841} C_DIS
LIN {X 53.157,Y 126.6177,Z 169,A 67.3342,B 9.7481,C 0.0808,E1 9.8121,E2 383.9753} C_DIS
LIN {X 56.5143,Y 125.156,Z 169,A 65.7,B 9.7481,C 0.0849,E1 9.8163,E2 385.6225} C_DIS
LIN {X 60.5504,Y 123.2532,Z 169,A 63.6854,B 9.748,C 0.0906,E1 9.8214,E2 387.6557} C_DIS
LIN {X 63.5078,Y 121.7561,Z 169,A 62.7793,B 9.748,C 0.0818,E1 9.8235,E2 388.5035} C_DIS
LIN {X 66.3674,Y 120.2231,Z 169,A 61.1532,B 9.748,C 0.0897,E1 9.8276,E2 390.1633} C_DIS
LIN {X 70.4317,Y 117.888,Z 169,A 59.2642,B 9.748,C 0.0911,E1 9.8321,E2 392.0442} C_DIS
LIN {X 74.1055,Y 115.6139,Z 169,A 57.4718,B 9.748,C 0.0936,E1 9.8364,E2 393.8356} C_DIS
LIN {X 77.4528,Y 113.3991,Z 169,A 55.836,B 9.748,C 0.0954,E1 9.8402,E2 395.4669} C_DIS
LIN {X 81.6633,Y 110.406,Z 169,A 53.5964,B 9.7479,C 0.1009,E1 9.8453,E2 397.7173} C_DIS
LIN {X 85.425,Y 107.521,Z 169,A 51.6854,B 9.7479,C 0.1028,E1 9.8494,E2 399.6204} C_DIS
LIN {X 89.3555,Y 104.2781,Z 169,A 49.5844,B 9.7479,C 0.1062,E1 9.8539,E2 401.7189} C_DIS
LIN {X 92.656,Y 101.3567,Z 169,A 47.795,B 9.7478,C 0.1086,E1 9.8576,E2 403.5028} C_DIS
LIN {X 95.7051,Y 98.4825,Z 169,A 46.2199,B 9.7478,C 0.108,E1 9.8608,E2 405.0572} C_DIS
LIN {X 98.1636,Y 96.0319,Z 169,A 44.6198,B 9.7478,C 0.1145,E1 9.864,E2 406.6764} C_DIS
LIN {X 102.6938,Y 91.1716,Z 169,A 41.9219,B 9.7477,C 0.1186,E1 9.8691,E2 409.3663} C_DIS
LIN {X 105.3349,Y 88.1067,Z 169,A 40.216,B 9.7477,C 0.1227,E1 9.8721,E2 411.0752} C_DIS
LIN {X 108.0824,Y 84.7137,Z 169,A 38.2675,B 9.7475,C 0.1298,E1 9.8756,E2 413.0402} C_DIS
LIN {X 111.153,Y 80.6425,Z 169,A 36.281,B 9.7475,C 0.1314,E1 9.8788,E2 415.0104} C_DIS
LIN {X 113.8391,Y 76.8043,Z 169,A 34.4044,B 9.7475,C 0.1342,E1 9.8818,E2 416.8783} C_DIS
LIN {X 116.0899,Y 73.3575,Z 169,A 32.6739,B 9.7475,C 0.1387,E1 9.8844,E2 418.6114} C_DIS
LIN {X 118.6029,Y 69.2222,Z 169,A 30.68,B 9.7473,C 0.1431,E1 9.8873,E2 420.6034} C_DIS
LIN {X 120.7413,Y 65.4209,Z 169,A 28.8231,B 9.7473,C 0.1486,E1 9.8898,E2 422.466} C_DIS
LIN {X 122.5343,Y 61.9927,Z 169,A 27.3243,B 9.7473,C 0.15,E1 9.8917,E2 423.9515} C_DIS
LIN {X 123.9942,Y 59.018,Z 169,A 25.9821,B 9.7473,C 0.1526,E1 9.8933,E2 425.2896} C_DIS
LIN {X 125.3896,Y 55.992,Z 169,A 24.5975,B 9.7471,C 0.1561,E1 9.8949,E2 426.6744} C_DIS
LIN {X 126.9701,Y 52.3134,Z 169,A 22.9892,B 9.7471,C 0.1591,E1 9.8966,E2 428.2762} C_DIS
LIN {X 128.1263,Y 49.411,Z 169,A 21.3802,B 9.7469,C 0.1699,E1 9.8983,E2 429.9241} C_DIS
LIN {X 129.3174,Y 46.2043,Z 169,A 20.3435,B 9.747,C 0.1644,E1 9.8993,E2 430.9133} C_DIS
LIN {X 130.2883,Y 43.3895,Z 169,A 19.0797,B 9.747,C 0.1683,E1 9.9004,E2 432.1808} C_DIS
LIN {X 131.339,Y 40.097,Z 169,A 17.6129,B 9.7469,C 0.1729,E1 9.9016,E2 433.6518} C_DIS
LIN {X 132.2947,Y 36.8216,Z 169,A 16.2297,B 9.7469,C 0.1759,E1 9.9027,E2 435.0311} C_DIS
LIN {X 133.2077,Y 33.3705,Z 169,A 14.7544,B 9.7467,C 0.1798,E1 9.9037,E2 436.5059} C_DIS
LIN {X 134.1742,Y 29.2417,Z 169,A 12.9855,B 9.7467,C 0.1848,E1 9.9048,E2 438.2763} C_DIS
LIN {X 134.8781,Y 25.8001,Z 169,A 11.5552,B 9.7466,C 0.1881,E1 9.9056,E2 439.7034} C_DIS
LIN {X 135.463,Y 22.5281,Z 169,A 10.185,B 9.7466,C 0.1917,E1 9.9062,E2 441.0727} C_DIS
LIN {X 136.0603,Y 18.5992,Z 169,A 8.6141,B 9.7465,C 0.1943,E1 9.9068,E2 442.6343} C_DIS
LIN {X 136.8091,Y 11.8804,Z 169,A 5.9948,B 9.7465,C 0.1976,E1 9.9076,E2 445.2309} C_DIS
LIN {X 137.0819,Y 8.15,Z 169,A 3.9587,B 9.7461,C 0.2137,E1 9.908,E2 447.3279} C_DIS
LIN {X 137.2466,Y 4.6535,Z 169,A 1.8957,B 9.7456,C 0.2324,E1 9.9082,E2 449.4671} C_DIS
LIN {X 137.3081,Y -2.0835,Z 169,A 0.295,B 9.7461,C 0.2114,E1 9.9082,E2 450.9197} C_DIS
LIN {X 137.0618,Y -8.4762,Z 169,A -2.5766,B 9.7458,C 0.2241,E1 9.9078,E2 453.8195} C_DIS
LIN {X 136.56,Y -14.4636,Z 169,A -5.0542,B 9.7457,C 0.2307,E1 9.9072,E2 456.2961} C_DIS
LIN {X 136.149,Y -17.9226,Z 169,A -6.4591,B 9.7457,C 0.2338,E1 9.9067,E2 457.6964} C_DIS
LIN {X 135.3605,Y -23.1427,Z 169,A -8.534,B 9.7455,C 0.237,E1 9.9058,E2 459.7574} C_DIS
LIN {X 134.8256,Y -26.0746,Z 169,A -9.9872,B 9.7453,C 0.2457,E1 9.9051,E2 461.2384} C_DIS
LIN {X 134.0046,Y -30.0136,Z 169,A -11.6396,B 9.7453,C 0.2499,E1 9.9041,E2 462.8892} C_DIS
LIN {X 132.9827,Y -34.2571,Z 169,A -13.3,B 9.7452,C 0.2512,E1 9.903,E2 464.5313} C_DIS
LIN {X 132.0287,Y -37.7722,Z 169,A -15.0706,B 9.7449,C 0.2616,E1 9.9016,E2 466.3351} C_DIS
LIN {X 130.7285,Y -42.0456,Z 169,A -16.62,B 9.7449,C 0.2592,E1 9.9004,E2 467.8469} C_DIS
LIN {X 129.6358,Y -45.303,Z 169,A -18.1015,B 9.7449,C 0.2644,E1 9.899,E2 469.336} C_DIS
LIN {X 127.7335,Y -50.4217,Z 169,A -20.336,B 9.7447,C 0.2696,E1 9.8968,E2 471.5675} C_DIS
LIN {X 126.1043,Y -54.3635,Z 169,A -22.0585,B 9.7446,C 0.2731,E1 9.895,E2 473.2846} C_DIS
LIN {X 124.7012,Y -57.509,Z 169,A -23.8808,B 9.7442,C 0.2862,E1 9.8928,E2 475.157} C_DIS
LIN {X 123.0088,Y -61.0457,Z 169,A -25.0913,B 9.7444,C 0.2804,E1 9.8914,E2 476.3158} C_DIS
Enddeposition()
END
